KUKA KRL program: MyProgram_281().src

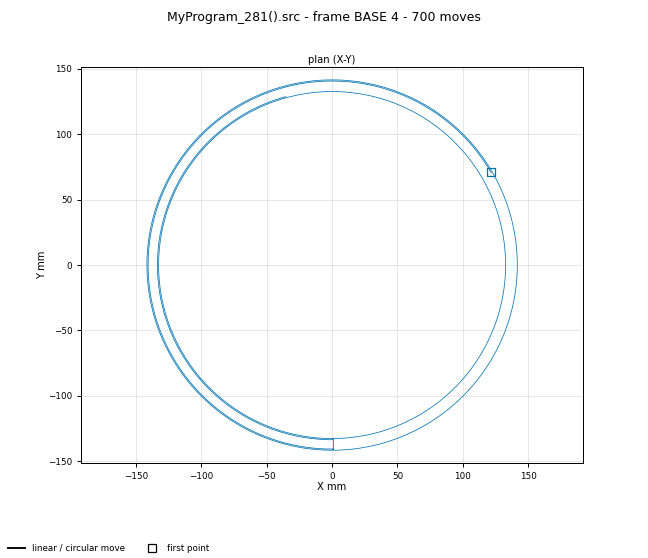
[picture p0: tool path of MyProgram_281().src in frame BASE 4, 700 of 700 moves have a stored position in this frame; points joined in program order, loops and branches not executed]
&ACCESS RVP
&REL 1
&PARAM TEMPLATE = C:\KRC\Roboter\Template\vorgabe
&PARAM EDITMASK = *
DEF MyProgram_281()
; ---- Setting reference (Base) ----
$BASE = BASE_DATA[4]

; --------------------------
; ---- Setting tool (TCP) ----
$TOOL = TOOL_DATA[3]
; --------------------------

$VEL.CP = VEL_APROX_PRINT
Startdeposition()
$VEL.CP = VEL_PRINT
LIN {X 121.5397,Y 70.8644,Z 173,A 32.0171,B 8.0887,C 0.1794,E1 8.2284,E2 419.8054} C_DIS
LIN {X 119.2507,Y 74.6518,Z 173,A 33.7721,B 8.0887,C 0.176,E1 8.2258,E2 418.0556} C_DIS
LIN {X 116.9146,Y 78.2591,Z 173,A 35.5172,B 8.0888,C 0.1719,E1 8.2231,E2 416.3103} C_DIS
LIN {X 114.3453,Y 81.9674,Z 173,A 37.3012,B 8.0889,C 0.1687,E1 8.2202,E2 414.5323} C_DIS
LIN {X 111.9951,Y 85.1512,Z 173,A 39.575,B 8.0893,C 0.1513,E1 8.2163,E2 412.1717} C_DIS
LIN {X 108.1696,Y 89.9605,Z 173,A 41.4044,B 8.0891,C 0.1597,E1 8.2132,E2 410.4289} C_DIS
LIN {X 105.5546,Y 93.0147,Z 173,A 43.0233,B 8.0891,C 0.1566,E1 8.2102,E2 408.8119} C_DIS
LIN {X 102.1646,Y 96.7261,Z 173,A 44.9523,B 8.0891,C 0.1547,E1 8.2066,E2 406.8974} C_DIS
LIN {X 99.1597,Y 99.804,Z 173,A 46.5834,B 8.0892,C 0.1536,E1 8.2034,E2 405.2813} C_DIS
LIN {X 93.6633,Y 104.9796,Z 173,A 49.7603,B 8.0894,C 0.1456,E1 8.1969,E2 402.0906} C_DIS
LIN {X 90.2461,Y 107.9313,Z 173,A 51.5389,B 8.0894,C 0.1434,E1 8.1931,E2 400.3193} C_DIS
LIN {X 86.802,Y 110.7199,Z 173,A 53.3455,B 8.0894,C 0.1401,E1 8.1891,E2 398.5122} C_DIS
LIN {X 83.1158,Y 113.5134,Z 173,A 55.2323,B 8.0895,C 0.1368,E1 8.1849,E2 396.6246} C_DIS
LIN {X 79.1384,Y 116.3216,Z 173,A 57.1673,B 8.0895,C 0.1345,E1 8.1805,E2 394.6955} C_DIS
LIN {X 75.4314,Y 118.7592,Z 173,A 58.9862,B 8.0895,C 0.1315,E1 8.1762,E2 392.8748} C_DIS
LIN {X 71.5988,Y 121.1084,Z 173,A 60.8066,B 8.0896,C 0.129,E1 8.1718,E2 391.0557} C_DIS
LIN {X 67.7143,Y 123.3224,Z 173,A 62.4595,B 8.0896,C 0.1297,E1 8.1679,E2 389.4242} C_DIS
LIN {X 62.8759,Y 125.8572,Z 173,A 64.811,B 8.0897,C 0.1244,E1 8.162,E2 387.0565} C_DIS
LIN {X 59.2274,Y 127.613,Z 173,A 66.3529,B 8.0897,C 0.1244,E1 8.1581,E2 385.5283} C_DIS
LIN {X 55.8685,Y 129.1187,Z 173,A 67.9786,B 8.0897,C 0.1202,E1 8.1539,E2 383.8865} C_DIS
LIN {X 51.5879,Y 130.8895,Z 173,A 69.7454,B 8.0897,C 0.1205,E1 8.1494,E2 382.1352} C_DIS
LIN {X 48.0453,Y 132.2298,Z 173,A 71.184,B 8.0897,C 0.121,E1 8.1457,E2 380.71} C_DIS
LIN {X 44.5635,Y 133.4431,Z 173,A 72.7767,B 8.0898,C 0.1179,E1 8.1414,E2 379.106} C_DIS
LIN {X 41.2024,Y 134.5189,Z 173,A 74.1193,B 8.0898,C 0.1184,E1 8.1379,E2 377.7757} C_DIS
LIN {X 38.0254,Y 135.4513,Z 173,A 75.499,B 8.0898,C 0.1168,E1 8.1342,E2 376.3921} C_DIS
LIN {X 35.189,Y 136.217,Z 173,A 77.1535,B 8.09,C 0.1073,E1 8.1296,E2 374.6794} C_DIS
LIN {X 31.0744,Y 137.2131,Z 173,A 78.431,B 8.0899,C 0.1146,E1 8.1262,E2 373.4594} C_DIS
LIN {X 27.0733,Y 138.0597,Z 173,A 80.1396,B 8.0899,C 0.1129,E1 8.1215,E2 371.7459} C_DIS
LIN {X 23.5323,Y 138.7061,Z 173,A 81.6734,B 8.0899,C 0.1109,E1 8.1173,E2 370.2038} C_DIS
LIN {X 18.8429,Y 139.4213,Z 173,A 83.3498,B 8.0899,C 0.1148,E1 8.1127,E2 368.5606} C_DIS
LIN {X 15.7013,Y 139.8103,Z 173,A 84.6671,B 8.0899,C 0.1139,E1 8.1091,E2 367.2401} C_DIS
LIN {X 12.7325,Y 140.1122,Z 173,A 86.1282,B 8.0899,C 0.1091,E1 8.1049,E2 365.7483} C_DIS
LIN {X 7.9682,Y 140.4636,Z 173,A 87.8716,B 8.0899,C 0.1124,E1 8.1001,E2 364.0314} C_DIS
LIN {X 4.257,Y 140.6239,Z 173,A 89.3394,B 8.0899,C 0.1131,E1 8.0961,E2 362.5699} C_DIS
LIN {X 1.4394,Y 140.6821,Z 173,A 90.4859,B 8.0899,C 0.1131,E1 8.0929,E2 361.4241} C_DIS
LIN {X -2.2697,Y 140.6696,Z 173,A 91.9938,B 8.0899,C 0.1131,E1 8.0887,E2 359.9172} C_DIS
LIN {X -5.6115,Y 140.5759,Z 173,A 93.5151,B 8.0899,C 0.1104,E1 8.0844,E2 358.3762} C_DIS
LIN {X -9.3168,Y 140.3806,Z 173,A 94.9136,B 8.0899,C 0.1127,E1 8.0805,E2 356.9929} C_DIS
LIN {X -12.9669,Y 140.0897,Z 173,A 96.3139,B 8.0899,C 0.1147,E1 8.0766,E2 355.6048} C_DIS
LIN {X -16.4487,Y 139.723,Z 173,A 97.8535,B 8.0899,C 0.1131,E1 8.0723,E2 354.0516} C_DIS
LIN {X -20.196,Y 139.2309,Z 173,A 99.5893,B 8.0899,C 0.1103,E1 8.0675,E2 352.2917} C_DIS
LIN {X -26.297,Y 138.2081,Z 173,A 102.423,B 8.0899,C 0.1062,E1 8.0596,E2 349.4193} C_DIS
LIN {X -30.692,Y 137.3005,Z 173,A 103.8767,B 8.0899,C 0.1138,E1 8.0557,E2 348.0146} C_DIS
LIN {X -35.3761,Y 136.1695,Z 173,A 105.8869,B 8.0899,C 0.1144,E1 8.0503,E2 345.9996} C_DIS
LIN {X -39.8029,Y 134.9399,Z 173,A 107.6544,B 8.0899,C 0.1176,E1 8.0456,E2 344.2465} C_DIS
LIN {X -44.0839,Y 133.6028,Z 173,A 109.4479,B 8.0898,C 0.1198,E1 8.0408,E2 342.4584} C_DIS
LIN {X -47.929,Y 132.2717,Z 173,A 111.3832,B 8.0898,C 0.1168,E1 8.0356,E2 340.4889} C_DIS
LIN {X -51.7917,Y 130.8101,Z 173,A 112.8658,B 8.0898,C 0.1219,E1 8.0318,E2 339.0331} C_DIS
LIN {X -55.5091,Y 129.2741,Z 173,A 114.4912,B 8.0898,C 0.124,E1 8.0277,E2 337.4105} C_DIS
LIN {X -61.4365,Y 126.5671,Z 173,A 117.2281,B 8.0897,C 0.1259,E1 8.0207,E2 334.6653} C_DIS
LIN {X -65.0696,Y 124.7357,Z 173,A 118.8403,B 8.0897,C 0.1288,E1 8.0167,E2 333.0599} C_DIS
LIN {X -68.2489,Y 123.0268,Z 173,A 120.467,B 8.0897,C 0.1283,E1 8.0127,E2 331.4146} C_DIS
LIN {X -72.3988,Y 120.632,Z 173,A 122.4005,B 8.0897,C 0.1315,E1 8.0081,E2 329.4851} C_DIS
LIN {X -76.3232,Y 118.1879,Z 173,A 124.3082,B 8.0896,C 0.134,E1 8.0036,E2 327.5758} C_DIS
LIN {X -80.2438,Y 115.5613,Z 173,A 126.0393,B 8.0895,C 0.1402,E1 7.9996,E2 325.8706} C_DIS
LIN {X -84.9117,Y 112.1763,Z 173,A 129.2567,B 8.0896,C 0.1303,E1 7.9922,E2 322.5441} C_DIS
LIN {X -89.5623,Y 108.4994,Z 173,A 130.8771,B 8.0893,C 0.1475,E1 7.9889,E2 321.0277} C_DIS
LIN {X -92.9813,Y 105.5841,Z 173,A 132.9319,B 8.0893,C 0.1475,E1 7.9845,E2 318.9459} C_DIS
LIN {X -95.7766,Y 103.055,Z 173,A 134.6016,B 8.0893,C 0.1483,E1 7.981,E2 317.2605} C_DIS
LIN {X -99.701,Y 99.2633,Z 173,A 136.5293,B 8.0891,C 0.1575,E1 7.9773,E2 315.3724} C_DIS
LIN {X -104.3128,Y 94.4052,Z 173,A 139.3278,B 8.0891,C 0.1622,E1 7.9719,E2 312.5678} C_DIS
LIN {X -109.1757,Y 88.7372,Z 173,A 142.5436,B 8.089,C 0.1663,E1 7.9661,E2 309.3328} C_DIS
LIN {X -111.9882,Y 85.1602,Z 173,A 144.3871,B 8.0889,C 0.1707,E1 7.9629,E2 307.4923} C_DIS
LIN {X -114.5373,Y 81.699,Z 173,A 146.118,B 8.0888,C 0.1751,E1 7.9601,E2 305.7656} C_DIS
LIN {X -116.8361,Y 78.3766,Z 173,A 147.8453,B 8.0888,C 0.1778,E1 7.9574,E2 304.0296} C_DIS
LIN {X -120.2813,Y 72.9789,Z 173,A 150.5347,B 8.0886,C 0.183,E1 7.9534,E2 301.3323} C_DIS
LIN {X -122.903,Y 68.4723,Z 173,A 152.688,B 8.0885,C 0.1879,E1 7.9504,E2 299.1773} C_DIS
LIN {X -125.091,Y 64.386,Z 173,A 154.5092,B 8.0884,C 0.1937,E1 7.948,E2 297.3665} C_DIS
LIN {X -126.5803,Y 61.4089,Z 173,A 156.0139,B 8.0884,C 0.195,E1 7.9462,E2 295.8442} C_DIS
LIN {X -128.0317,Y 58.3219,Z 173,A 157.4645,B 8.0883,C 0.1978,E1 7.9445,E2 294.3871} C_DIS
LIN {X -129.6212,Y 54.695,Z 173,A 158.9373,B 8.0881,C 0.2042,E1 7.9429,E2 292.9338} C_DIS
LIN {X -130.9965,Y 51.3126,Z 173,A 160.2682,B 8.0879,C 0.2105,E1 7.9415,E2 291.6243} C_DIS
LIN {X -132.2272,Y 48.0524,Z 173,A 161.9677,B 8.0879,C 0.2102,E1 7.9398,E2 289.8903} C_DIS
LIN {X -133.4973,Y 44.4008,Z 173,A 163.4771,B 8.0879,C 0.2155,E1 7.9385,E2 288.3909} C_DIS
LIN {X -134.5688,Y 41.0391,Z 173,A 164.8901,B 8.0877,C 0.2198,E1 7.9373,E2 286.9823} C_DIS
LIN {X -135.4878,Y 37.8948,Z 173,A 166.2428,B 8.0877,C 0.2233,E1 7.9363,E2 285.6285} C_DIS
LIN {X -136.2722,Y 34.9715,Z 173,A 167.6133,B 8.0876,C 0.2246,E1 7.9353,E2 284.2416} C_DIS
LIN {X -137.0675,Y 31.7118,Z 173,A 169.0149,B 8.0875,C 0.228,E1 7.9344,E2 282.8367} C_DIS
LIN {X -138.4552,Y 24.9642,Z 173,A 171.7558,B 8.0872,C 0.2369,E1 7.9329,E2 280.1069} C_DIS
LIN {X -139.392,Y 19.0614,Z 173,A 174.3063,B 8.0871,C 0.2422,E1 7.9318,E2 277.5439} C_DIS
LIN {X -139.9884,Y 14.0225,Z 173,A 176.6134,B 8.087,C 0.2445,E1 7.9311,E2 275.2077} C_DIS
LIN {X -140.3173,Y 10.2038,Z 173,A 178.5693,B 8.087,C 0.243,E1 7.9307,E2 273.2019} C_DIS
LIN {X -140.5888,Y 5.2818,Z 173,A -179.9247,B 8.0866,C 0.2564,E1 7.9305,E2 271.7629} C_DIS
LIN {X -140.6787,Y -1.7183,Z 173,A -176.9036,B 8.0864,C 0.2621,E1 7.9305,E2 268.7225} C_DIS
LIN {X -140.5167,Y -6.9375,Z 173,A -174.8865,B 8.0862,C 0.2698,E1 7.9307,E2 266.7214} C_DIS
LIN {X -140.2633,Y -10.9436,Z 173,A -173.1133,B 8.0862,C 0.2725,E1 7.9311,E2 264.9317} C_DIS
LIN {X -139.341,Y -19.4256,Z 173,A -169.8202,B 8.0857,C 0.2852,E1 7.9321,E2 261.6652} C_DIS
LIN {X -138.8167,Y -22.8693,Z 173,A -168.246,B 8.0857,C 0.2868,E1 7.9328,E2 260.072} C_DIS
LIN {X -138.2199,Y -26.2355,Z 173,A -166.7828,B 8.0855,C 0.2897,E1 7.9336,E2 258.6007} C_DIS
LIN {X -137.4925,Y -29.8133,Z 173,A -165.3249,B 8.0853,C 0.2943,E1 7.9344,E2 257.1477} C_DIS
LIN {X -136.7395,Y -33.0954,Z 173,A -163.9364,B 8.0853,C 0.2979,E1 7.9353,E2 255.7579} C_DIS
LIN {X -135.9183,Y -36.3208,Z 173,A -162.5627,B 8.0851,C 0.3014,E1 7.9363,E2 254.3829} C_DIS
LIN {X -134.9268,Y -39.8475,Z 173,A -161.0054,B 8.085,C 0.3045,E1 7.9375,E2 252.8183} C_DIS
LIN {X -133.6154,Y -44.0459,Z 173,A -159.2293,B 8.0848,C 0.3096,E1 7.939,E2 251.0454} C_DIS
LIN {X -132.2087,Y -48.1038,Z 173,A -157.2964,B 8.0848,C 0.3115,E1 7.9408,E2 249.0898} C_DIS
LIN {X -130.5376,Y -52.468,Z 173,A -155.6934,B 8.0843,C 0.3212,E1 7.9424,E2 247.5271} C_DIS
LIN {X -129.2717,Y -55.5146,Z 173,A -154.1083,B 8.0843,C 0.321,E1 7.9441,E2 245.9115} C_DIS
LIN {X -127.8562,Y -58.7014,Z 173,A -152.6637,B 8.0843,C 0.3243,E1 7.9458,E2 244.4646} C_DIS
LIN {X -126.333,Y -61.9114,Z 173,A -151.2786,B 8.084,C 0.3289,E1 7.9475,E2 243.0884} C_DIS
LIN {X -124.5763,Y -65.3731,Z 173,A -148.4644,B 8.0846,C 0.3135,E1 7.9514,E2 240.1127} C_DIS
LIN {X -120.64,Y -72.3853,Z 173,A -146.1641,B 8.0837,C 0.337,E1 7.9544,E2 237.9432} C_DIS
LIN {X -117.8769,Y -76.8022,Z 173,A -144.0223,B 8.0835,C 0.3417,E1 7.9576,E2 235.7998} C_DIS
LIN {X -115.2733,Y -80.6578,Z 173,A -142.085,B 8.0833,C 0.3454,E1 7.9607,E2 233.8579} C_DIS
LIN {X -112.6344,Y -84.3036,Z 173,A -140.2391,B 8.0832,C 0.3494,E1 7.9638,E2 232.0111} C_DIS
LIN {X -109.7952,Y -87.9698,Z 173,A -138.3153,B 8.083,C 0.353,E1 7.9671,E2 230.0834} C_DIS
LIN {X -106.8869,Y -91.4814,Z 173,A -136.1315,B 8.083,C 0.3517,E1 7.9711,E2 227.8573} C_DIS
LIN {X -104.2877,Y -94.4328,Z 173,A -134.8234,B 8.0827,C 0.3598,E1 7.9735,E2 226.5884} C_DIS
LIN {X -101.5037,Y -97.4195,Z 173,A -133.1573,B 8.0826,C 0.3631,E1 7.9767,E2 224.9224} C_DIS
LIN {X -98.6922,Y -100.2665,Z 173,A -131.3687,B 8.0826,C 0.3637,E1 7.9803,E2 223.1134} C_DIS
LIN {X -94.8602,Y -103.9,Z 173,A -129.2725,B 8.0823,C 0.3686,E1 7.9846,E2 221.025} C_DIS
LIN {X -91.3696,Y -106.9821,Z 173,A -127.3587,B 8.0822,C 0.3718,E1 7.9886,E2 219.1092} C_DIS
LIN {X -87.741,Y -109.9773,Z 173,A -125.4408,B 8.082,C 0.3751,E1 7.9928,E2 217.1915} C_DIS
LIN {X -83.5306,Y -113.2086,Z 173,A -123.1789,B 8.082,C 0.377,E1 7.9978,E2 214.9167} C_DIS
LIN {X -79.4321,Y -116.1209,Z 173,A -121.217,B 8.0817,C 0.3816,E1 8.0023,E2 212.9664} C_DIS
LIN {X -75.8907,Y -118.4655,Z 173,A -119.466,B 8.0817,C 0.3838,E1 8.0064,E2 211.2128} C_DIS
LIN {X -71.8963,Y -120.9315,Z 173,A -117.5578,B 8.0815,C 0.3865,E1 8.011,E2 209.3051} C_DIS
LIN {X -69.3467,Y -122.412,Z 173,A -115.7889,B 8.0819,C 0.3784,E1 8.0155,E2 207.4609} C_DIS
LIN {X -64.8654,Y -124.8429,Z 173,A -114.2083,B 8.0813,C 0.3895,E1 8.0192,E2 205.9462} C_DIS
LIN {X -61.0098,Y -126.771,Z 173,A -112.5189,B 8.0812,C 0.3927,E1 8.0234,E2 204.2655} C_DIS
LIN {X -56.6312,Y -128.7889,Z 173,A -110.574,B 8.0811,C 0.3952,E1 8.0284,E2 202.323} C_DIS
LIN {X -53.3702,Y -130.1739,Z 173,A -108.9867,B 8.0811,C 0.3941,E1 8.0325,E2 200.7165} C_DIS
LIN {X -49.8269,Y -131.5693,Z 173,A -107.6282,B 8.0809,C 0.3989,E1 8.036,E2 199.3831} C_DIS
LIN {X -46.9077,Y -132.6399,Z 173,A -106.18,B 8.0809,C 0.3968,E1 8.0398,E2 197.9108} C_DIS
LIN {X -43.0184,Y -133.9493,Z 173,A -104.614,B 8.0809,C 0.4,E1 8.044,E2 196.3583} C_DIS
LIN {X -38.913,Y -135.2004,Z 173,A -102.5335,B 8.0811,C 0.3952,E1 8.0497,E2 194.2334} C_DIS
LIN {X -35.4651,Y -136.1465,Z 173,A -101.3993,B 8.0807,C 0.4019,E1 8.0526,E2 193.1416} C_DIS
LIN {X -31.503,Y -137.1152,Z 173,A -99.6866,B 8.0807,C 0.4019,E1 8.0573,E2 191.4217} C_DIS
LIN {X -28.5134,Y -137.7687,Z 173,A -98.4424,B 8.0807,C 0.4026,E1 8.0607,E2 190.1774} C_DIS
LIN {X -25.6225,Y -138.3364,Z 173,A -97.109,B 8.0808,C 0.4006,E1 8.0644,E2 188.826} C_DIS
LIN {X -21.893,Y -138.9743,Z 173,A -95.8468,B 8.0805,C 0.4062,E1 8.0678,E2 187.6003} C_DIS
LIN {X -18.5725,Y -139.4567,Z 173,A -94.2702,B 8.0807,C 0.4028,E1 8.0722,E2 185.9953} C_DIS
LIN {X -14.0852,Y -139.9824,Z 173,A -92.475,B 8.0807,C 0.404,E1 8.0772,E2 184.2054} C_DIS
LIN {X -10.485,Y -140.2967,Z 173,A -90.9975,B 8.0807,C 0.404,E1 8.0813,E2 182.7265} C_DIS
LIN {X -6.2607,Y -140.5505,Z 173,A -89.1335,B 8.0807,C 0.4014,E1 8.0865,E2 180.8431} C_DIS
LIN {X -1.5063,Y -140.6817,Z 173,A -87.3668,B 8.0807,C 0.4045,E1 8.0914,E2 179.0982} C_DIS
LIN {X 0.9966,Y -140.684,Z 173,A -86.7203,B 8.0803,C 0.4113,E1 8.0931,E2 178.5006} C_DIS
Enddeposition()
LIN {X 0.9966,Y -140.684,Z 173,A -86.7203,B 8.0803,C 0.4113,E1 8.0931,E2 178.5006} C_DIS
Startdeposition()
$VEL.CP = VEL_PRINT
LIN {X 0.0008,Y -141.5985,Z 173,A -87.3284,B 8.0796,C 0.42,E1 8.091,E2 179.1698} C_DIS
LIN {X -2.9523,Y -141.5669,Z 173,A -88.5344,B 8.0796,C 0.4203,E1 8.0877,E2 180.3779} C_DIS
LIN {X -6.4248,Y -141.4522,Z 173,A -90.091,B 8.0795,C 0.4231,E1 8.0833,E2 181.9551} C_DIS
LIN {X -10.4048,Y -141.2135,Z 173,A -91.574,B 8.0796,C 0.4205,E1 8.0792,E2 183.4214} C_DIS
LIN {X -13.8781,Y -140.915,Z 173,A -92.979,B 8.0796,C 0.4202,E1 8.0753,E2 184.8262} C_DIS
LIN {X -17.1895,Y -140.5496,Z 173,A -94.3385,B 8.0796,C 0.4202,E1 8.0715,E2 186.1877} C_DIS
LIN {X -20.7709,Y -140.0665,Z 173,A -95.7933,B 8.0796,C 0.4196,E1 8.0675,E2 187.642} C_DIS
LIN {X -24.2041,Y -139.5142,Z 173,A -97.2155,B 8.0796,C 0.4194,E1 8.0635,E2 189.0667} C_DIS
LIN {X -27.6244,Y -138.8767,Z 173,A -98.6204,B 8.0797,C 0.4187,E1 8.0597,E2 190.4716} C_DIS
LIN {X -31.0173,Y -138.1581,Z 173,A -99.9098,B 8.0798,C 0.416,E1 8.0562,E2 191.7464} C_DIS
LIN {X -33.8951,Y -137.4813,Z 173,A -101.2277,B 8.0798,C 0.4175,E1 8.0526,E2 193.0806} C_DIS
LIN {X -37.2579,Y -136.6086,Z 173,A -102.6325,B 8.0798,C 0.4166,E1 8.0488,E2 194.4856} C_DIS
LIN {X -40.3664,Y -135.7216,Z 173,A -104.1154,B 8.0798,C 0.4188,E1 8.0448,E2 195.9918} C_DIS
LIN {X -44.9118,Y -134.2847,Z 173,A -105.97,B 8.0798,C 0.416,E1 8.0399,E2 197.837} C_DIS
LIN {X -48.8467,Y -132.9065,Z 173,A -107.5933,B 8.08,C 0.4134,E1 8.0356,E2 199.4522} C_DIS
LIN {X -52.0928,Y -131.668,Z 173,A -109.0108,B 8.08,C 0.4123,E1 8.0319,E2 200.8713} C_DIS
LIN {X -56.2644,Y -129.9373,Z 173,A -110.896,B 8.08,C 0.4114,E1 8.027,E2 202.7642} C_DIS
LIN {X -59.7557,Y -128.3697,Z 173,A -112.4081,B 8.0802,C 0.4091,E1 8.0232,E2 204.2716} C_DIS
LIN {X -63.4258,Y -126.599,Z 173,A -114.0734,B 8.0802,C 0.4075,E1 8.019,E2 205.9391} C_DIS
LIN {X -66.7353,Y -124.8858,Z 173,A -115.6997,B 8.0802,C 0.4076,E1 8.015,E2 207.5811} C_DIS
LIN {X -70.5472,Y -122.7731,Z 173,A -117.4889,B 8.0804,C 0.4057,E1 8.0106,E2 209.3736} C_DIS
LIN {X -74.5003,Y -120.415,Z 173,A -119.3629,B 8.0804,C 0.4033,E1 8.0061,E2 211.2489} C_DIS
LIN {X -78.1616,Y -118.0713,Z 173,A -121.1386,B 8.0806,C 0.401,E1 8.002,E2 213.0266} C_DIS
LIN {X -82.0256,Y -115.4206,Z 173,A -123.0413,B 8.0807,C 0.3981,E1 7.9976,E2 214.9299} C_DIS
LIN {X -85.7396,Y -112.6889,Z 173,A -124.8747,B 8.0809,C 0.3945,E1 7.9935,E2 216.7588} C_DIS
LIN {X -89.1541,Y -110.0073,Z 173,A -126.7136,B 8.0809,C 0.3929,E1 7.9895,E2 218.6081} C_DIS
LIN {X -92.6824,Y -107.0516,Z 173,A -128.5779,B 8.0812,C 0.3896,E1 7.9855,E2 220.4723} C_DIS
LIN {X -96.1818,Y -103.9191,Z 173,A -130.4624,B 8.0813,C 0.3858,E1 7.9816,E2 222.3542} C_DIS
LIN {X -99.3281,Y -100.9155,Z 173,A -132.2779,B 8.0815,C 0.3833,E1 7.978,E2 224.1765} C_DIS
LIN {X -102.5166,Y -97.6746,Z 173,A -134.0126,B 8.0817,C 0.3779,E1 7.9746,E2 225.8968} C_DIS
LIN {X -104.91,Y -95.0991,Z 173,A -135.5902,B 8.0817,C 0.3775,E1 7.9716,E2 227.4942} C_DIS
LIN {X -107.9521,Y -91.6313,Z 173,A -137.4853,B 8.0819,C 0.374,E1 7.9681,E2 229.3923} C_DIS
LIN {X -110.9324,Y -88,Z 173,A -139.3449,B 8.0821,C 0.3692,E1 7.9649,E2 231.2458} C_DIS
LIN {X -113.578,Y -84.5575,Z 173,A -141.1682,B 8.0822,C 0.3663,E1 7.9618,E2 233.077} C_DIS
LIN {X -116.2656,Y -80.8224,Z 173,A -143.0817,B 8.0824,C 0.3628,E1 7.9587,E2 234.9964} C_DIS
LIN {X -118.6886,Y -77.2204,Z 173,A -144.8629,B 8.0826,C 0.3591,E1 7.956,E2 236.7799} C_DIS
LIN {X -121.136,Y -73.3214,Z 173,A -146.749,B 8.0827,C 0.355,E1 7.9532,E2 238.668} C_DIS
LIN {X -123.4918,Y -69.2801,Z 173,A -148.6629,B 8.0829,C 0.3506,E1 7.9505,E2 240.5836} C_DIS
LIN {X -125.567,Y -65.4406,Z 173,A -150.397,B 8.0831,C 0.3457,E1 7.9483,E2 242.3126} C_DIS
LIN {X -126.9801,Y -62.6533,Z 173,A -151.7113,B 8.0832,C 0.3433,E1 7.9466,E2 243.6326} C_DIS
LIN {X -128.6243,Y -59.205,Z 173,A -153.2596,B 8.0834,C 0.3393,E1 7.9448,E2 245.1802} C_DIS
LIN {X -130.1442,Y -55.7861,Z 173,A -154.7693,B 8.0836,C 0.3353,E1 7.9431,E2 246.6885} C_DIS
LIN {X -131.4752,Y -52.5722,Z 173,A -156.1988,B 8.0837,C 0.3319,E1 7.9416,E2 248.1199} C_DIS
LIN {X -132.7228,Y -49.3375,Z 173,A -157.6704,B 8.0838,C 0.3292,E1 7.9401,E2 249.5994} C_DIS
LIN {X -134.2854,Y -44.9097,Z 173,A -159.5572,B 8.084,C 0.3239,E1 7.9384,E2 251.4832} C_DIS
LIN {X -135.3463,Y -41.6032,Z 173,A -161.0737,B 8.0841,C 0.3217,E1 7.9371,E2 253.0131} C_DIS
LIN {X -136.4655,Y -37.7722,Z 173,A -162.6285,B 8.0843,C 0.3164,E1 7.9359,E2 254.559} C_DIS
LIN {X -137.3538,Y -34.4031,Z 173,A -164.062,B 8.0845,C 0.3128,E1 7.9349,E2 255.9945} C_DIS
LIN {X -138.1566,Y -31.0238,Z 173,A -165.4411,B 8.0846,C 0.3085,E1 7.9341,E2 257.369} C_DIS
LIN {X -138.7726,Y -28.1359,Z 173,A -166.711,B 8.0847,C 0.3063,E1 7.9334,E2 258.6477} C_DIS
LIN {X -139.4213,Y -24.7232,Z 173,A -168.1406,B 8.0849,C 0.3027,E1 7.9326,E2 260.0793} C_DIS
LIN {X -139.987,Y -21.2903,Z 173,A -169.5528,B 8.0849,C 0.2987,E1 7.932,E2 261.491} C_DIS
LIN {X -140.4695,Y -17.8361,Z 173,A -171.0016,B 8.0851,C 0.2953,E1 7.9315,E2 262.9435} C_DIS
LIN {X -140.865,Y -14.3923,Z 173,A -172.4437,B 8.0852,C 0.2919,E1 7.931,E2 264.3895} C_DIS
LIN {X -141.1748,Y -10.9356,Z 173,A -173.9987,B 8.0853,C 0.2901,E1 7.9307,E2 265.9627} C_DIS
LIN {X -141.425,Y -6.9652,Z 173,A -175.5055,B 8.0855,C 0.2839,E1 7.9304,E2 267.4548} C_DIS
LIN {X -141.5537,Y -3.5022,Z 173,A -176.9238,B 8.0857,C 0.2801,E1 7.9304,E2 268.8739} C_DIS
LIN {X -141.5999,Y -0.016,Z 173,A -178.3743,B 8.0857,C 0.2766,E1 7.9303,E2 270.3284} C_DIS
LIN {X -141.5207,Y 4.6893,Z 173,A 179.6709,B 8.0859,C 0.2719,E1 7.9304,E2 272.2879} C_DIS
LIN {X -141.3313,Y 8.6596,Z 173,A 178.0397,B 8.0861,C 0.2676,E1 7.9307,E2 273.9205} C_DIS
LIN {X -141.0751,Y 12.1397,Z 173,A 176.6126,B 8.0862,C 0.2637,E1 7.931,E2 275.3483} C_DIS
LIN {X -140.7367,Y 15.5848,Z 173,A 175.187,B 8.0863,C 0.2601,E1 7.9314,E2 276.7757} C_DIS
LIN {X -140.3111,Y 19.0453,Z 173,A 173.7549,B 8.0864,C 0.2564,E1 7.9319,E2 278.2092} C_DIS
LIN {X -139.8046,Y 22.468,Z 173,A 172.3118,B 8.0865,C 0.253,E1 7.9325,E2 279.6566} C_DIS
LIN {X -139.2133,Y 25.8774,Z 173,A 170.8827,B 8.0867,C 0.2494,E1 7.9332,E2 281.0881} C_DIS
LIN {X -138.5378,Y 29.2766,Z 173,A 169.5536,B 8.0868,C 0.2444,E1 7.9339,E2 282.4064} C_DIS
LIN {X -137.8858,Y 32.2095,Z 173,A 168.2359,B 8.0868,C 0.2425,E1 7.9348,E2 283.736} C_DIS
LIN {X -137.0534,Y 35.5868,Z 173,A 166.7963,B 8.087,C 0.239,E1 7.9358,E2 285.1784} C_DIS
LIN {X -136.1394,Y 38.9383,Z 173,A 165.2183,B 8.087,C 0.2376,E1 7.937,E2 286.777} C_DIS
LIN {X -135.0545,Y 42.5444,Z 173,A 163.6509,B 8.0871,C 0.2341,E1 7.9383,E2 288.3484} C_DIS
LIN {X -133.4964,Y 47.2108,Z 173,A 161.7841,B 8.0873,C 0.2268,E1 7.9399,E2 290.1975} C_DIS
LIN {X -132.2979,Y 50.4719,Z 173,A 160.351,B 8.0874,C 0.2233,E1 7.9413,E2 291.6327} C_DIS
LIN {X -131.0192,Y 53.7033,Z 173,A 158.6858,B 8.0874,C 0.2234,E1 7.9431,E2 293.3294} C_DIS
LIN {X -129.0903,Y 58.1828,Z 173,A 156.8718,B 8.0876,C 0.2158,E1 7.9451,E2 295.1212} C_DIS
LIN {X -127.2479,Y 62.1104,Z 173,A 155.23,B 8.0878,C 0.2095,E1 7.9471,E2 296.7467} C_DIS
LIN {X -125.9654,Y 64.6709,Z 173,A 153.8757,B 8.0878,C 0.2095,E1 7.9488,E2 298.1247} C_DIS
LIN {X -123.7569,Y 68.8059,Z 173,A 151.9893,B 8.0879,C 0.2044,E1 7.9513,E2 300.008} C_DIS
LIN {X -121.5879,Y 72.5696,Z 173,A 150.1547,B 8.0879,C 0.2012,E1 7.9539,E2 301.8506} C_DIS
LIN {X -119.1717,Y 76.4728,Z 173,A 148.31,B 8.0881,C 0.1964,E1 7.9567,E2 303.6918} C_DIS
LIN {X -116.7581,Y 80.1093,Z 173,A 146.46,B 8.0881,C 0.1934,E1 7.9596,E2 305.5507} C_DIS
LIN {X -114.0944,Y 83.8595,Z 173,A 144.5675,B 8.0883,C 0.1895,E1 7.9627,E2 307.4453} C_DIS
LIN {X -111.4706,Y 87.3171,Z 173,A 142.783,B 8.0883,C 0.1859,E1 7.9657,E2 309.2317} C_DIS
LIN {X -108.5516,Y 90.9203,Z 173,A 140.8956,B 8.0884,C 0.1819,E1 7.9691,E2 311.1186} C_DIS
LIN {X -105.5581,Y 94.3792,Z 173,A 139.0023,B 8.0885,C 0.1785,E1 7.9726,E2 313.0156} C_DIS
LIN {X -102.6012,Y 97.5862,Z 173,A 137.1886,B 8.0885,C 0.1755,E1 7.976,E2 314.8337} C_DIS
LIN {X -99.515,Y 100.7316,Z 173,A 135.4599,B 8.0887,C 0.171,E1 7.9794,E2 316.5539} C_DIS
LIN {X -96.5769,Y 103.5512,Z 173,A 133.7939,B 8.0887,C 0.1679,E1 7.9828,E2 318.2206} C_DIS
LIN {X -93.3587,Y 106.4622,Z 173,A 131.9544,B 8.0887,C 0.1659,E1 7.9867,E2 320.069} C_DIS
LIN {X -89.8361,Y 109.4509,Z 173,A 130.0589,B 8.0888,C 0.1628,E1 7.9907,E2 321.9661} C_DIS
LIN {X -86.4521,Y 112.1433,Z 173,A 128.2813,B 8.0889,C 0.1601,E1 7.9946,E2 323.7456} C_DIS
LIN {X -82.7628,Y 114.8931,Z 173,A 126.3907,B 8.0889,C 0.1573,E1 7.9989,E2 325.6382} C_DIS
LIN {X -78.8844,Y 117.5895,Z 173,A 124.5314,B 8.089,C 0.1534,E1 8.0032,E2 327.4893} C_DIS
LIN {X -75.2389,Y 119.9551,Z 173,A 122.7046,B 8.089,C 0.1517,E1 8.0075,E2 329.3232} C_DIS
LIN {X -71.3046,Y 122.3347,Z 173,A 120.8109,B 8.0891,C 0.1495,E1 8.012,E2 331.2195} C_DIS
LIN {X -67.2852,Y 124.5903,Z 173,A 118.946,B 8.0891,C 0.1469,E1 8.0166,E2 333.0828} C_DIS
LIN {X -63.6672,Y 126.4763,Z 173,A 117.431,B 8.0892,C 0.1424,E1 8.0203,E2 334.5793} C_DIS
LIN {X -60.7819,Y 127.8867,Z 173,A 116.0719,B 8.0892,C 0.1418,E1 8.0238,E2 335.9449} C_DIS
LIN {X -57.6143,Y 129.3446,Z 173,A 114.6219,B 8.0892,C 0.1407,E1 8.0274,E2 337.3988} C_DIS
LIN {X -54.1942,Y 130.8149,Z 173,A 113.1381,B 8.0892,C 0.1386,E1 8.0313,E2 338.8786} C_DIS
LIN {X -50.978,Y 132.1013,Z 173,A 111.6788,B 8.0893,C 0.1381,E1 8.0351,E2 340.3441} C_DIS
LIN {X -47.2193,Y 133.4934,Z 173,A 109.9184,B 8.0893,C 0.1388,E1 8.0397,E2 342.1209} C_DIS
LIN {X -43.26,Y 134.8259,Z 173,A 108.3938,B 8.0893,C 0.1345,E1 8.0437,E2 343.6233} C_DIS
LIN {X -39.4413,Y 135.9924,Z 173,A 106.771,B 8.0893,C 0.1332,E1 8.0481,E2 345.2458} C_DIS
LIN {X -36.0943,Y 136.9189,Z 173,A 105.2913,B 8.0893,C 0.1334,E1 8.0521,E2 346.7341} C_DIS
LIN {X -31.8757,Y 137.962,Z 173,A 103.5209,B 8.0894,C 0.1324,E1 8.0569,E2 348.5048} C_DIS
LIN {X -28.1671,Y 138.7663,Z 173,A 102.052,B 8.0894,C 0.1304,E1 8.0609,E2 349.9643} C_DIS
LIN {X -24.7634,Y 139.4141,Z 173,A 100.6464,B 8.0894,C 0.1297,E1 8.0647,E2 351.3696} C_DIS
LIN {X -21.3335,Y 139.9803,Z 173,A 99.2799,B 8.0894,C 0.1283,E1 8.0685,E2 352.7301} C_DIS
LIN {X -17.851,Y 140.4676,Z 173,A 97.8181,B 8.0894,C 0.1285,E1 8.0725,E2 354.1961} C_DIS
LIN {X -14.8389,Y 140.8169,Z 173,A 96.5366,B 8.0894,C 0.129,E1 8.0761,E2 355.4838} C_DIS
LIN {X -10.9413,Y 141.1744,Z 173,A 94.8643,B 8.0894,C 0.1302,E1 8.0808,E2 357.1666} C_DIS
LIN {X -6.9546,Y 141.4255,Z 173,A 93.3776,B 8.0894,C 0.1276,E1 8.0849,E2 358.636} C_DIS
LIN {X -3.4759,Y 141.5545,Z 173,A 91.9802,B 8.0894,C 0.1273,E1 8.0888,E2 360.0313} C_DIS
LIN {X -0.0037,Y 141.5985,Z 173,A 90.5893,B 8.0894,C 0.127,E1 8.0927,E2 361.4198} C_DIS
LIN {X 2.9503,Y 141.5669,Z 173,A 89.3828,B 8.0894,C 0.1272,E1 8.096,E2 362.6272} C_DIS
LIN {X 6.4229,Y 141.4523,Z 173,A 88.0062,B 8.0894,C 0.1268,E1 8.0999,E2 363.9995} C_DIS
LIN {X 10.4159,Y 141.2127,Z 173,A 86.3436,B 8.0894,C 0.1279,E1 8.1045,E2 365.667} C_DIS
LIN {X 13.8739,Y 140.9154,Z 173,A 84.9459,B 8.0894,C 0.1282,E1 8.1084,E2 367.0634} C_DIS
LIN {X 17.3249,Y 140.5335,Z 173,A 83.5468,B 8.0894,C 0.1285,E1 8.1123,E2 368.4612} C_DIS
LIN {X 20.7727,Y 140.0662,Z 173,A 82.141,B 8.0894,C 0.129,E1 8.1162,E2 369.8663} C_DIS
LIN {X 24.2085,Y 139.5134,Z 173,A 80.7176,B 8.0894,C 0.13,E1 8.1201,E2 371.2913} C_DIS
LIN {X 27.6173,Y 138.8781,Z 173,A 79.3225,B 8.0894,C 0.1306,E1 8.1239,E2 372.685} C_DIS
LIN {X 31.0091,Y 138.16,Z 173,A 78.0496,B 8.0894,C 0.129,E1 8.1273,E2 373.9409} C_DIS
LIN {X 33.8918,Y 137.4821,Z 173,A 76.7425,B 8.0894,C 0.1318,E1 8.1309,E2 375.2617} C_DIS
LIN {X 37.2334,Y 136.6152,Z 173,A 75.3502,B 8.0894,C 0.1328,E1 8.1347,E2 376.653} C_DIS
LIN {X 41.1056,Y 135.4986,Z 173,A 73.7236,B 8.0894,C 0.134,E1 8.139,E2 378.2788} C_DIS
LIN {X 44.9102,Y 134.2852,Z 173,A 72.0442,B 8.0894,C 0.1366,E1 8.1435,E2 379.966} C_DIS
LIN {X 48.8461,Y 132.9067,Z 173,A 70.4393,B 8.0894,C 0.1366,E1 8.1477,E2 381.5602} C_DIS
LIN {X 52.0935,Y 131.6677,Z 173,A 69.0389,B 8.0894,C 0.138,E1 8.1514,E2 382.9598} C_DIS
LIN {X 55.2644,Y 130.368,Z 173,A 67.6052,B 8.0893,C 0.1404,E1 8.1551,E2 384.3993} C_DIS
LIN {X 58.1475,Y 129.1061,Z 173,A 66.396,B 8.0893,C 0.1407,E1 8.1581,E2 385.6002} C_DIS
LIN {X 61.3132,Y 127.6329,Z 173,A 64.9404,B 8.0893,C 0.1432,E1 8.1618,E2 387.0612} C_DIS
LIN {X 65.1957,Y 125.6957,Z 173,A 63.1609,B 8.0892,C 0.146,E1 8.1663,E2 388.8438} C_DIS
LIN {X 69.2618,Y 123.5021,Z 173,A 61.3074,B 8.0892,C 0.1482,E1 8.1708,E2 390.6953} C_DIS
LIN {X 73.3198,Y 121.1369,Z 173,A 59.4409,B 8.0891,C 0.1503,E1 8.1753,E2 392.5576} C_DIS
LIN {X 76.997,Y 118.8336,Z 173,A 57.6959,B 8.0891,C 0.1528,E1 8.1794,E2 394.3013} C_DIS
LIN {X 80.815,Y 116.2707,Z 173,A 55.8446,B 8.089,C 0.1556,E1 8.1836,E2 396.1517} C_DIS
LIN {X 84.5584,Y 113.5774,Z 173,A 53.9974,B 8.089,C 0.1584,E1 8.1878,E2 397.9968} C_DIS
LIN {X 88.0013,Y 110.9314,Z 173,A 52.2498,B 8.0889,C 0.1613,E1 8.1916,E2 399.7435} C_DIS
LIN {X 91.6265,Y 107.9562,Z 173,A 50.438,B 8.0889,C 0.1631,E1 8.1955,E2 401.5448} C_DIS
LIN {X 94.8379,Y 105.147,Z 173,A 48.7244,B 8.0888,C 0.1661,E1 8.1991,E2 403.2571} C_DIS
LIN {X 98.0085,Y 102.1975,Z 173,A 47.0248,B 8.0888,C 0.1685,E1 8.2025,E2 404.9505} C_DIS
LIN {X 100.7366,Y 99.5101,Z 173,A 45.4619,B 8.0887,C 0.1719,E1 8.2056,E2 406.5156} C_DIS
LIN {X 103.5606,Y 96.5668,Z 173,A 43.7986,B 8.0886,C 0.1756,E1 8.2088,E2 408.1811} C_DIS
LIN {X 106.6406,Y 93.1544,Z 173,A 41.9441,B 8.0885,C 0.1795,E1 8.2123,E2 410.0355} C_DIS
LIN {X 109.5062,Y 89.7685,Z 173,A 40.1682,B 8.0885,C 0.183,E1 8.2154,E2 411.8097} C_DIS
LIN {X 112.4634,Y 86.0345,Z 173,A 38.3566,B 8.0884,C 0.185,E1 8.2185,E2 413.6072} C_DIS
LIN {X 114.9114,Y 82.7375,Z 173,A 36.6167,B 8.0883,C 0.1904,E1 8.2214,E2 415.3579} C_DIS
LIN {X 117.5913,Y 78.8818,Z 173,A 34.8133,B 8.0882,C 0.1929,E1 8.2242,E2 417.1498} C_DIS
LIN {X 119.9533,Y 75.2417,Z 173,A 33.0329,B 8.0881,C 0.1977,E1 8.2269,E2 418.9342} C_DIS
LIN {X 122.3336,Y 71.3065,Z 173,A 31.1849,B 8.088,C 0.202,E1 8.2295,E2 420.7816} C_DIS
LIN {X 124.5907,Y 67.2844,Z 173,A 29.3643,B 8.0879,C 0.2058,E1 8.232,E2 422.5974} C_DIS
LIN {X 126.4775,Y 63.6649,Z 173,A 27.8401,B 8.0879,C 0.2073,E1 8.2339,E2 424.1061} C_DIS
LIN {X 128.0049,Y 60.5346,Z 173,A 26.3573,B 8.0877,C 0.2125,E1 8.2357,E2 425.5991} C_DIS
LIN {X 129.9343,Y 56.2714,Z 173,A 24.513,B 8.0877,C 0.2164,E1 8.2378,E2 427.4382} C_DIS
LIN {X 131.4657,Y 52.5955,Z 173,A 23.003,B 8.0875,C 0.2186,E1 8.2394,E2 428.9362} C_DIS
LIN {X 132.7224,Y 49.3384,Z 173,A 21.5724,B 8.0875,C 0.2227,E1 8.2408,E2 430.3701} C_DIS
LIN {X 134.285,Y 44.911,Z 173,A 19.7492,B 8.0873,C 0.2263,E1 8.2425,E2 432.1846} C_DIS
LIN {X 135.3462,Y 41.6036,Z 173,A 18.284,B 8.0872,C 0.2314,E1 8.2437,E2 433.6586} C_DIS
LIN {X 136.4681,Y 37.7631,Z 173,A 16.7782,B 8.0872,C 0.2335,E1 8.2448,E2 435.151} C_DIS
LIN {X 137.3585,Y 34.3844,Z 173,A 15.3905,B 8.087,C 0.2369,E1 8.2458,E2 436.5363} C_DIS
LIN {X 138.1594,Y 31.0115,Z 173,A 14.0601,B 8.087,C 0.2393,E1 8.2466,E2 437.8584} C_DIS
LIN {X 138.7737,Y 28.1309,Z 173,A 12.8391,B 8.0868,C 0.2432,E1 8.2473,E2 439.084} C_DIS
LIN {X 139.3908,Y 24.8932,Z 173,A 11.5045,B 8.0868,C 0.247,E1 8.248,E2 440.4198} C_DIS
LIN {X 139.9855,Y 21.3,Z 173,A 10.0861,B 8.0866,C 0.25,E1 8.2486,E2 441.8323} C_DIS
LIN {X 140.4663,Y 17.8607,Z 173,A 8.71,B 8.0866,C 0.2534,E1 8.2491,E2 443.2057} C_DIS
LIN {X 140.8645,Y 14.3964,Z 173,A 7.3124,B 8.0864,C 0.2572,E1 8.2496,E2 444.6029} C_DIS
LIN {X 141.1747,Y 10.9366,Z 173,A 5.8101,B 8.0862,C 0.2633,E1 8.2499,E2 446.1189} C_DIS
LIN {X 141.4255,Y 6.9545,Z 173,A 4.3526,B 8.0862,C 0.2646,E1 8.2501,E2 447.5573} C_DIS
LIN {X 141.5542,Y 3.4847,Z 173,A 2.8703,B 8.086,C 0.2703,E1 8.2503,E2 449.051} C_DIS
LIN {X 141.5957,Y -0.7174,Z 173,A 1.2301,B 8.0859,C 0.2739,E1 8.2503,E2 450.6848} C_DIS
LIN {X 141.5207,Y -4.6903,Z 173,A -0.2955,B 8.0858,C 0.2768,E1 8.2502,E2 452.2012} C_DIS
LIN {X 141.3677,Y -8.0688,Z 173,A -1.7661,B 8.0856,C 0.283,E1 8.2499,E2 453.6863} C_DIS
LIN {X 141.0747,Y -12.1452,Z 173,A -3.2472,B 8.0856,C 0.284,E1 8.2496,E2 455.1464} C_DIS
LIN {X 140.7341,Y -15.6089,Z 173,A -4.6256,B 8.0854,C 0.2874,E1 8.2492,E2 456.5222} C_DIS
LIN {X 140.3099,Y -19.0538,Z 173,A -6.003,B 8.0853,C 0.2909,E1 8.2487,E2 457.8975} C_DIS
LIN {X 139.8013,Y -22.4888,Z 173,A -7.4056,B 8.0851,C 0.2949,E1 8.2481,E2 459.301} C_DIS
LIN {X 139.2074,Y -25.9084,Z 173,A -8.7833,B 8.0851,C 0.2983,E1 8.2475,E2 460.6766} C_DIS
LIN {X 138.6684,Y -28.6479,Z 173,A -9.8961,B 8.0849,C 0.3012,E1 8.2468,E2 461.7882} C_DIS
LIN {X 137.8864,Y -32.2065,Z 173,A -11.3281,B 8.0848,C 0.3045,E1 8.246,E2 463.2162} C_DIS
LIN {X 137.056,Y -35.5765,Z 173,A -12.7094,B 8.0847,C 0.3079,E1 8.245,E2 464.5958} C_DIS
LIN {X 136.1424,Y -38.9276,Z 173,A -14.2231,B 8.0844,C 0.3142,E1 8.2439,E2 466.1251} C_DIS
LIN {X 135.0248,Y -42.6375,Z 173,A -15.7647,B 8.0843,C 0.318,E1 8.2426,E2 467.6648} C_DIS
LIN {X 133.4962,Y -47.2113,Z 173,A -17.5546,B 8.0842,C 0.3199,E1 8.241,E2 469.4354} C_DIS
LIN {X 132.2963,Y -50.476,Z 173,A -18.9396,B 8.0841,C 0.3233,E1 8.2396,E2 470.819} C_DIS
LIN {X 131.0182,Y -53.7059,Z 173,A -20.5457,B 8.0837,C 0.3314,E1 8.2379,E2 472.4528} C_DIS
LIN {X 129.0978,Y -58.1662,Z 173,A -22.2551,B 8.0837,C 0.3312,E1 8.236,E2 474.1305} C_DIS
LIN {X 127.6337,Y -61.3116,Z 173,A -23.6902,B 8.0836,C 0.3356,E1 8.2343,E2 475.5712} C_DIS
LIN {X 125.7117,Y -65.1652,Z 173,A -25.4552,B 8.0834,C 0.3406,E1 8.2321,E2 477.3409} C_DIS
LIN {X 123.4998,Y -69.2658,Z 173,A -27.298,B 8.0832,C 0.3446,E1 8.2296,E2 479.1801} C_DIS
LIN {X 121.1392,Y -73.316,Z 173,A -29.1526,B 8.083,C 0.3485,E1 8.227,E2 481.031} C_DIS
LIN {X 118.8297,Y -77.003,Z 173,A -30.8871,B 8.0829,C 0.3523,E1 8.2244,E2 482.7639} C_DIS
LIN {X 116.2746,Y -80.8094,Z 173,A -32.7227,B 8.0827,C 0.3564,E1 8.2215,E2 484.5988} C_DIS
LIN {X 113.5927,Y -84.5379,Z 173,A -34.5545,B 8.0825,C 0.3603,E1 8.2185,E2 486.4289} C_DIS
LIN {X 110.9488,Y -87.9794,Z 173,A -36.3033,B 8.0823,C 0.3643,E1 8.2155,E2 488.1785} C_DIS
LIN {X 108.0432,Y -91.5242,Z 173,A -38.0946,B 8.0822,C 0.3672,E1 8.2123,E2 489.9633} C_DIS
LIN {X 105.0971,Y -94.8929,Z 173,A -39.8593,B 8.0821,C 0.3703,E1 8.209,E2 491.7237} C_DIS
LIN {X 102.1393,Y -98.0694,Z 173,A -41.5822,B 8.0819,C 0.3734,E1 8.2057,E2 493.4439} C_DIS
LIN {X 99.3241,Y -100.9194,Z 173,A -43.2451,B 8.0817,C 0.3777,E1 8.2024,E2 495.1139} C_DIS
LIN {X 96.1843,Y -103.9168,Z 173,A -44.9937,B 8.0816,C 0.3811,E1 8.1988,E2 496.8631} C_DIS
LIN {X 92.6912,Y -107.044,Z 173,A -46.8512,B 8.0814,C 0.3841,E1 8.195,E2 498.7171} C_DIS
LIN {X 89.1563,Y -110.0055,Z 173,A -48.7037,B 8.0813,C 0.3874,E1 8.191,E2 500.5697} C_DIS
LIN {X 85.7439,Y -112.6856,Z 173,A -50.4422,B 8.0811,C 0.3903,E1 8.1871,E2 502.3074} C_DIS
LIN {X 82.2509,Y -115.2595,Z 173,A -52.1665,B 8.081,C 0.3928,E1 8.1832,E2 504.0292} C_DIS
LIN {X 78.8832,Y -117.5903,Z 173,A -53.7541,B 8.081,C 0.3942,E1 8.1796,E2 505.6091} C_DIS
LIN {X 75.2475,Y -119.9496,Z 173,A -55.5403,B 8.0808,C 0.3978,E1 8.1754,E2 507.4012} C_DIS
LIN {X 71.3168,Y -122.3277,Z 173,A -57.3987,B 8.0806,C 0.4007,E1 8.1709,E2 509.261} C_DIS
LIN {X 67.2883,Y -124.5886,Z 173,A -59.234,B 8.0806,C 0.4028,E1 8.1664,E2 511.0934} C_DIS
LIN {X 63.6652,Y -126.4774,Z 173,A -60.7754,B 8.0806,C 0.4028,E1 8.1626,E2 512.6214} C_DIS
LIN {X 60.5414,Y -128.0017,Z 173,A -62.2591,B 8.0803,C 0.4063,E1 8.1589,E2 514.1164} C_DIS
LIN {X 56.2818,Y -129.9298,Z 173,A -64.1233,B 8.0803,C 0.4082,E1 8.1541,E2 515.9784} C_DIS
LIN {X 52.5796,Y -131.4722,Z 173,A -65.6525,B 8.0803,C 0.4082,E1 8.1502,E2 517.4965} C_DIS
LIN {X 49.3421,Y -132.7211,Z 173,A -67.0906,B 8.0801,C 0.4105,E1 8.1464,E2 518.9402} C_DIS
LIN {X 44.9193,Y -134.2822,Z 173,A -68.9306,B 8.0801,C 0.4114,E1 8.1416,E2 520.7739} C_DIS
LIN {X 41.6018,Y -135.3468,Z 173,A -70.4163,B 8.0799,C 0.4143,E1 8.1376,E2 522.2707} C_DIS
LIN {X 37.7687,Y -136.4665,Z 173,A -71.9384,B 8.0799,C 0.4139,E1 8.1335,E2 523.7815} C_DIS
LIN {X 34.3942,Y -137.3561,Z 173,A -73.3396,B 8.0799,C 0.4149,E1 8.1297,E2 525.1822} C_DIS
LIN {X 31.0215,Y -138.1571,Z 173,A -74.6857,B 8.0799,C 0.4149,E1 8.1261,E2 526.5217} C_DIS
LIN {X 28.1381,Y -138.7722,Z 173,A -75.9252,B 8.0799,C 0.4166,E1 8.1227,E2 527.7681} C_DIS
LIN {X 24.7294,Y -139.4201,Z 173,A -77.3215,B 8.0798,C 0.4174,E1 8.1188,E2 529.1643} C_DIS
LIN {X 21.3039,Y -139.9849,Z 173,A -78.7181,B 8.0798,C 0.418,E1 8.115,E2 530.5607} C_DIS
LIN {X 17.8626,Y -140.466,Z 173,A -80.1158,B 8.0798,C 0.4186,E1 8.1111,E2 531.9581} C_DIS
LIN {X 14.3981,Y -140.8644,Z 173,A -81.5336,B 8.0797,C 0.4193,E1 8.1072,E2 533.3777} C_DIS
LIN {X 10.9385,Y -141.1746,Z 173,A -83.0598,B 8.0795,C 0.4221,E1 8.1029,E2 534.9206} C_DIS
LIN {X 6.9583,Y -141.4254,Z 173,A -84.5416,B 8.0796,C 0.42,E1 8.0988,E2 536.3858} C_DIS
LIN {X 3.5575,Y -141.5522,Z 173,A -85.9138,B 8.0796,C 0.4202,E1 8.095,E2 537.758} C_DIS
LIN {X 1.0025,Y -141.5919,Z 173,A -86.6713,B 8.0799,C 0.4152,E1 8.093,E2 538.4792} C_DIS
Enddeposition()
LIN {X 0.9609,Y -132.6531,Z 174,A -86.8217,B 7.8952,C 0.3729,E1 7.9067,E2 538.3641} C_DIS
Startdeposition()
$VEL.CP = VEL_PRINT
LIN {X 3.5384,Y -132.6117,Z 174,A -85.4392,B 7.8955,C 0.3681,E1 7.9107,E2 536.9479} C_DIS
LIN {X 6.5007,Y -132.4995,Z 174,A -84.1106,B 7.8955,C 0.367,E1 7.9144,E2 535.6127} C_DIS
LIN {X 9.7566,Y -132.2995,Z 174,A -82.7613,B 7.8955,C 0.3676,E1 7.9182,E2 534.27} C_DIS
LIN {X 13.5559,Y -131.9658,Z 174,A -81.1804,B 7.8955,C 0.3681,E1 7.9225,E2 532.6965} C_DIS
LIN {X 16.9055,Y -131.5775,Z 174,A -79.8457,B 7.8954,C 0.3695,E1 7.9262,E2 531.376} C_DIS
LIN {X 19.4578,Y -131.2258,Z 174,A -78.4735,B 7.8956,C 0.3644,E1 7.9301,E2 529.971} C_DIS
LIN {X 22.9482,Y -130.6594,Z 174,A -77.1207,B 7.8956,C 0.3666,E1 7.9338,E2 528.6389} C_DIS
LIN {X 26.1646,Y -130.0531,Z 174,A -75.6205,B 7.8956,C 0.3641,E1 7.9379,E2 527.1271} C_DIS
LIN {X 29.0672,Y -129.4358,Z 174,A -74.273,B 7.8957,C 0.362,E1 7.9416,E2 525.7706} C_DIS
LIN {X 32.5097,Y -128.6134,Z 174,A -72.8269,B 7.8957,C 0.3622,E1 7.9455,E2 524.3337} C_DIS
LIN {X 35.6508,Y -127.7783,Z 174,A -71.431,B 7.8957,C 0.3611,E1 7.9493,E2 522.9378} C_DIS
LIN {X 39.3639,Y -126.6849,Z 174,A -69.609,B 7.896,C 0.3568,E1 7.9542,E2 521.096} C_DIS
LIN {X 43.4371,Y -125.3454,Z 174,A -67.9306,B 7.896,C 0.358,E1 7.9586,E2 519.4378} C_DIS
LIN {X 46.4958,Y -124.2432,Z 174,A -66.6072,B 7.896,C 0.358,E1 7.962,E2 518.1232} C_DIS
LIN {X 49.2601,Y -123.1739,Z 174,A -65.199,B 7.896,C 0.3541,E1 7.9657,E2 516.6982} C_DIS
LIN {X 52.5282,Y -121.8156,Z 174,A -63.7504,B 7.8961,C 0.3537,E1 7.9694,E2 515.2584} C_DIS
LIN {X 55.2378,Y -120.6119,Z 174,A -62.4842,B 7.8961,C 0.3523,E1 7.9726,E2 513.993} C_DIS
LIN {X 58.4338,Y -119.0957,Z 174,A -60.9597,B 7.8963,C 0.3503,E1 7.9765,E2 512.4676} C_DIS
LIN {X 61.3534,Y -117.6185,Z 174,A -59.6166,B 7.8963,C 0.3496,E1 7.9798,E2 511.1321} C_DIS
LIN {X 64.1418,Y -116.1232,Z 174,A -58.2767,B 7.8963,C 0.3481,E1 7.9831,E2 509.7944} C_DIS
LIN {X 66.7445,Y -114.6474,Z 174,A -56.9304,B 7.8965,C 0.3451,E1 7.9864,E2 508.4403} C_DIS
LIN {X 69.4956,Y -113.0006,Z 174,A -55.4972,B 7.8966,C 0.342,E1 7.9898,E2 506.9998} C_DIS
LIN {X 73.0679,Y -110.7242,Z 174,A -53.8777,B 7.8966,C 0.3429,E1 7.9935,E2 505.4048} C_DIS
LIN {X 75.0508,Y -109.3898,Z 174,A -52.6532,B 7.8968,C 0.3375,E1 7.9964,E2 504.1556} C_DIS
LIN {X 77.7176,Y -107.5116,Z 174,A -51.3426,B 7.8968,C 0.3368,E1 7.9994,E2 502.8559} C_DIS
LIN {X 80.8479,Y -105.1783,Z 174,A -49.6486,B 7.897,C 0.3336,E1 8.0032,E2 501.1594} C_DIS
LIN {X 84.0476,Y -102.639,Z 174,A -47.8822,B 7.8971,C 0.3302,E1 8.007,E2 499.3911} C_DIS
LIN {X 87.2606,Y -99.9216,Z 174,A -46.0051,B 7.8973,C 0.3255,E1 8.011,E2 497.5049} C_DIS
LIN {X 90.3246,Y -97.1608,Z 174,A -44.2828,B 7.8974,C 0.323,E1 8.0145,E2 495.7882} C_DIS
LIN {X 92.558,Y -95.0364,Z 174,A -42.9023,B 7.8976,C 0.3193,E1 8.0173,E2 494.4004} C_DIS
LIN {X 95.6132,Y -91.9622,Z 174,A -41.0747,B 7.8976,C 0.3162,E1 8.0209,E2 492.5766} C_DIS
LIN {X 98.3947,Y -88.9791,Z 174,A -39.3603,B 7.8978,C 0.3132,E1 8.0241,E2 490.8663} C_DIS
LIN {X 101.3796,Y -85.5632,Z 174,A -37.4681,B 7.8979,C 0.3101,E1 8.0275,E2 488.9804} C_DIS
LIN {X 104.0784,Y -82.2594,Z 174,A -35.699,B 7.898,C 0.3073,E1 8.0306,E2 487.2186} C_DIS
LIN {X 106.5557,Y -79.0234,Z 174,A -33.9536,B 7.8982,C 0.3034,E1 8.0335,E2 485.4733} C_DIS
LIN {X 108.765,Y -75.9538,Z 174,A -32.4826,B 7.8982,C 0.3026,E1 8.0359,E2 484.0208} C_DIS
LIN {X 110.4637,Y -73.4615,Z 174,A -31.1547,B 7.8984,C 0.299,E1 8.038,E2 482.6884} C_DIS
LIN {X 112.2359,Y -70.7238,Z 174,A -29.7192,B 7.8985,C 0.2949,E1 8.0401,E2 481.2482} C_DIS
LIN {X 113.9345,Y -67.9536,Z 174,A -28.3321,B 7.8986,C 0.2917,E1 8.0421,E2 479.8617} C_DIS
LIN {X 115.5801,Y -65.1154,Z 174,A -27.0164,B 7.8986,C 0.2901,E1 8.0439,E2 478.5571} C_DIS
LIN {X 116.9988,Y -62.531,Z 174,A -25.6698,B 7.8989,C 0.2854,E1 8.0458,E2 477.2002} C_DIS
LIN {X 118.4918,Y -59.6513,Z 174,A -24.2958,B 7.8989,C 0.2822,E1 8.0475,E2 475.8282} C_DIS
LIN {X 120.0296,Y -56.4952,Z 174,A -22.823,B 7.8991,C 0.2791,E1 8.0493,E2 474.3592} C_DIS
LIN {X 121.26,Y -53.7995,Z 174,A -21.5588,B 7.8991,C 0.276,E1 8.0507,E2 473.0956} C_DIS
LIN {X 122.6727,Y -50.4984,Z 174,A -20.0384,B 7.8993,C 0.2724,E1 8.0524,E2 471.5775} C_DIS
LIN {X 123.7686,Y -47.7461,Z 174,A -18.7834,B 7.8994,C 0.2694,E1 8.0536,E2 470.3241} C_DIS
LIN {X 124.9019,Y -44.6973,Z 174,A -17.3754,B 7.8995,C 0.2655,E1 8.055,E2 468.9144} C_DIS
LIN {X 126.1735,Y -40.9746,Z 174,A -15.7632,B 7.8996,C 0.2625,E1 8.0564,E2 467.3113} C_DIS
LIN {X 127.3232,Y -37.2432,Z 174,A -14.037,B 7.8998,C 0.257,E1 8.0578,E2 465.5785} C_DIS
LIN {X 128.2656,Y -33.8575,Z 174,A -12.5923,B 7.8999,C 0.2542,E1 8.0588,E2 464.1413} C_DIS
LIN {X 129.1004,Y -30.5237,Z 174,A -11.1518,B 7.9,C 0.2509,E1 8.0598,E2 462.7047} C_DIS
LIN {X 129.7876,Y -27.4551,Z 174,A -9.7649,B 7.9002,C 0.2465,E1 8.0606,E2 461.3131} C_DIS
LIN {X 130.4186,Y -24.2835,Z 174,A -8.4035,B 7.9002,C 0.2432,E1 8.0613,E2 459.9547} C_DIS
LIN {X 131.0216,Y -20.7823,Z 174,A -6.9107,B 7.9004,C 0.2396,E1 8.062,E2 458.4655} C_DIS
LIN {X 131.491,Y -17.5658,Z 174,A -5.5342,B 7.9004,C 0.2361,E1 8.0625,E2 457.091} C_DIS
LIN {X 131.9263,Y -13.9235,Z 174,A -4.0523,B 7.9005,C 0.2336,E1 8.063,E2 455.6202} C_DIS
LIN {X 132.1934,Y -11.1018,Z 174,A -2.8379,B 7.9006,C 0.2303,E1 8.0633,E2 454.4058} C_DIS
LIN {X 132.4274,Y -7.8379,Z 174,A -1.4394,B 7.9008,C 0.2265,E1 8.0636,E2 453.0079} C_DIS
LIN {X 132.5694,Y -4.8791,Z 174,A -0.1515,B 7.9008,C 0.2226,E1 8.0637,E2 451.7178} C_DIS
LIN {X 132.6543,Y -1.2569,Z 174,A 1.2235,B 7.9008,C 0.2219,E1 8.0637,E2 450.3647} C_DIS
LIN {X 132.6455,Y 1.9089,Z 174,A 2.7477,B 7.9011,C 0.2148,E1 8.0637,E2 448.8201} C_DIS
LIN {X 132.5585,Y 5.1584,Z 174,A 4.1585,B 7.9011,C 0.2106,E1 8.0637,E2 447.4072} C_DIS
LIN {X 132.3912,Y 8.4261,Z 174,A 5.5202,B 7.9013,C 0.2076,E1 8.0634,E2 446.0507} C_DIS
LIN {X 132.048,Y 12.7143,Z 174,A 7.3658,B 7.9013,C 0.2025,E1 8.0629,E2 444.2049} C_DIS
LIN {X 131.6629,Y 16.2319,Z 174,A 8.8183,B 7.9015,C 0.1997,E1 8.0625,E2 442.7605} C_DIS
LIN {X 131.178,Y 19.772,Z 174,A 10.3489,B 7.9015,C 0.1955,E1 8.0619,E2 441.2302} C_DIS
LIN {X 130.656,Y 22.9672,Z 174,A 11.6301,B 7.9016,C 0.1938,E1 8.0613,E2 439.9621} C_DIS
LIN {X 130.0538,Y 26.1608,Z 174,A 13.1006,B 7.9017,C 0.1886,E1 8.0605,E2 438.4824} C_DIS
LIN {X 129.4365,Y 29.0639,Z 174,A 14.4332,B 7.9018,C 0.184,E1 8.0597,E2 437.1427} C_DIS
LIN {X 128.6113,Y 32.5181,Z 174,A 15.8635,B 7.9019,C 0.1817,E1 8.0587,E2 435.7238} C_DIS
LIN {X 127.7752,Y 35.662,Z 174,A 17.2435,B 7.9019,C 0.1783,E1 8.0577,E2 434.3459} C_DIS
LIN {X 126.8558,Y 38.8056,Z 174,A 18.6316,B 7.9021,C 0.1749,E1 8.0566,E2 432.9599} C_DIS
LIN {X 125.7327,Y 42.3049,Z 174,A 20.2283,B 7.9021,C 0.1704,E1 8.0552,E2 431.3611} C_DIS
LIN {X 124.2522,Y 46.472,Z 174,A 21.9966,B 7.9022,C 0.1681,E1 8.0536,E2 429.6087} C_DIS
LIN {X 123.0543,Y 49.5568,Z 174,A 23.467,B 7.9022,C 0.1634,E1 8.052,E2 428.1323} C_DIS
LIN {X 121.8127,Y 52.5348,Z 174,A 24.844,B 7.9024,C 0.1601,E1 8.0505,E2 426.7564} C_DIS
LIN {X 120.6096,Y 55.2429,Z 174,A 26.0996,B 7.9024,C 0.1572,E1 8.0491,E2 425.5031} C_DIS
LIN {X 119.091,Y 58.4432,Z 174,A 27.6044,B 7.9024,C 0.1537,E1 8.0473,E2 424.0003} C_DIS
LIN {X 117.6192,Y 61.3519,Z 174,A 28.9491,B 7.9025,C 0.1514,E1 8.0456,E2 422.6625} C_DIS
LIN {X 116.2139,Y 63.9781,Z 174,A 30.254,B 7.9026,C 0.1478,E1 8.0438,E2 421.3548} C_DIS
LIN {X 114.6101,Y 66.809,Z 174,A 31.6473,B 7.9026,C 0.1445,E1 8.0419,E2 419.9621} C_DIS
LIN {X 112.9381,Y 69.5975,Z 174,A 33.0731,B 7.9027,C 0.1407,E1 8.0398,E2 418.5331} C_DIS
LIN {X 111.1996,Y 72.3424,Z 174,A 34.4505,B 7.9027,C 0.1378,E1 8.0377,E2 417.1581} C_DIS
LIN {X 109.3918,Y 75.0479,Z 174,A 35.789,B 7.9028,C 0.1357,E1 8.0356,E2 415.827} C_DIS
LIN {X 107.5075,Y 77.7233,Z 174,A 37.204,B 7.9028,C 0.1324,E1 8.0333,E2 414.4112} C_DIS
LIN {X 105.092,Y 80.9604,Z 174,A 39.0354,B 7.903,C 0.1268,E1 8.0302,E2 412.5686} C_DIS
LIN {X 102.4951,Y 84.2237,Z 174,A 40.81,B 7.903,C 0.1233,E1 8.0271,E2 410.7964} C_DIS
LIN {X 99.8224,Y 87.3743,Z 174,A 42.5669,B 7.903,C 0.1199,E1 8.0239,E2 409.0422} C_DIS
LIN {X 96.8512,Y 90.6571,Z 174,A 44.3871,B 7.9031,C 0.1176,E1 8.0205,E2 407.2325} C_DIS
LIN {X 94.1235,Y 93.4854,Z 174,A 45.8925,B 7.9031,C 0.1178,E1 8.0176,E2 405.7495} C_DIS
LIN {X 91.9616,Y 95.6138,Z 174,A 47.4319,B 7.9032,C 0.1109,E1 8.0145,E2 404.1823} C_DIS
LIN {X 88.5865,Y 98.7481,Z 174,A 49.3247,B 7.9032,C 0.1088,E1 8.0106,E2 402.3005} C_DIS
LIN {X 85.5222,Y 101.414,Z 174,A 51.0543,B 7.9032,C 0.106,E1 8.0069,E2 400.5735} C_DIS
LIN {X 82.2606,Y 104.0774,Z 174,A 52.8199,B 7.9032,C 0.1037,E1 8.0031,E2 398.8139} C_DIS
LIN {X 79.0205,Y 106.5579,Z 174,A 54.5725,B 7.9033,C 0.1009,E1 7.9992,E2 397.0622} C_DIS
LIN {X 76.1756,Y 108.6101,Z 174,A 55.9917,B 7.9033,C 0.1001,E1 7.996,E2 395.6542} C_DIS
LIN {X 73.459,Y 110.4653,Z 174,A 57.3872,B 7.9033,C 0.0983,E1 7.9928,E2 394.2616} C_DIS
LIN {X 70.7284,Y 112.233,Z 174,A 58.8273,B 7.9034,C 0.0955,E1 7.9894,E2 392.8172} C_DIS
LIN {X 67.9589,Y 113.9313,Z 174,A 60.2158,B 7.9034,C 0.0937,E1 7.986,E2 391.4303} C_DIS
LIN {X 65.1447,Y 115.5636,Z 174,A 61.5424,B 7.9034,C 0.0931,E1 7.9828,E2 390.1131} C_DIS
LIN {X 62.547,Y 116.9902,Z 174,A 63.0439,B 7.9034,C 0.0874,E1 7.9791,E2 388.5851} C_DIS
LIN {X 59.6377,Y 118.4987,Z 174,A 64.3077,B 7.9034,C 0.0883,E1 7.976,E2 387.3394} C_DIS
LIN {X 56.456,Y 120.0483,Z 174,A 65.8028,B 7.9035,C 0.087,E1 7.9722,E2 385.8484} C_DIS
LIN {X 53.7569,Y 121.2791,Z 174,A 67.072,B 7.9035,C 0.0857,E1 7.969,E2 384.5806} C_DIS
LIN {X 50.5027,Y 122.6709,Z 174,A 68.5908,B 7.9035,C 0.0842,E1 7.9651,E2 383.0632} C_DIS
LIN {X 47.7434,Y 123.7696,Z 174,A 69.8619,B 7.9035,C 0.083,E1 7.9618,E2 381.7935} C_DIS
LIN {X 44.6961,Y 124.9024,Z 174,A 71.3002,B 7.9035,C 0.0811,E1 7.958,E2 380.3513} C_DIS
LIN {X 41.018,Y 126.1596,Z 174,A 73.0975,B 7.9035,C 0.0775,E1 7.9532,E2 378.5402} C_DIS
LIN {X 36.9725,Y 127.4025,Z 174,A 74.7409,B 7.9035,C 0.0792,E1 7.9489,E2 376.9191} C_DIS
LIN {X 33.8592,Y 128.2651,Z 174,A 76.1287,B 7.9035,C 0.0783,E1 7.9451,E2 375.5325} C_DIS
LIN {X 29.9671,Y 129.2302,Z 174,A 77.989,B 7.9036,C 0.0749,E1 7.94,E2 373.6574} C_DIS
LIN {X 25.8777,Y 130.1114,Z 174,A 79.6487,B 7.9036,C 0.0764,E1 7.9355,E2 372.0156} C_DIS
LIN {X 22.6777,Y 130.7078,Z 174,A 81.1376,B 7.9036,C 0.0743,E1 7.9314,E2 370.5173} C_DIS
LIN {X 19.185,Y 131.2648,Z 174,A 82.5893,B 7.9036,C 0.0749,E1 7.9274,E2 369.0751} C_DIS
LIN {X 15.5065,Y 131.7495,Z 174,A 84.097,B 7.9036,C 0.0759,E1 7.9233,E2 367.5791} C_DIS
LIN {X 12.3477,Y 132.0832,Z 174,A 85.4945,B 7.9036,C 0.0751,E1 7.9194,E2 366.1791} C_DIS
LIN {X 9.7585,Y 132.2994,Z 174,A 86.7167,B 7.9036,C 0.0732,E1 7.916,E2 364.9454} C_DIS
LIN {X 6.5128,Y 132.4989,Z 174,A 88.0662,B 7.9036,C 0.0739,E1 7.9122,E2 363.6031} C_DIS
LIN {X 3.2641,Y 132.6194,Z 174,A 89.5103,B 7.9036,C 0.0731,E1 7.9082,E2 362.1548} C_DIS
LIN {X 0.0164,Y 132.6608,Z 174,A 90.9832,B 7.9036,C 0.072,E1 7.9041,E2 360.6742} C_DIS
LIN {X -3.5439,Y 132.6116,Z 174,A 92.421,B 7.9036,C 0.0737,E1 7.9001,E2 359.249} C_DIS
LIN {X -6.5062,Y 132.4993,Z 174,A 93.751,B 7.9036,C 0.0731,E1 7.8963,E2 357.9137} C_DIS
LIN {X -9.752,Y 132.2999,Z 174,A 95.1031,B 7.9036,C 0.0742,E1 7.8926,E2 356.5685} C_DIS
LIN {X -13.0004,Y 132.0206,Z 174,A 96.509,B 7.9036,C 0.0746,E1 7.8887,E2 355.1637} C_DIS
LIN {X -16.241,Y 131.6618,Z 174,A 97.9164,B 7.9036,C 0.0751,E1 7.8848,E2 353.7571} C_DIS
LIN {X -19.4633,Y 131.225,Z 174,A 99.4199,B 7.9036,C 0.0741,E1 7.8806,E2 352.2428} C_DIS
LIN {X -22.956,Y 130.658,Z 174,A 100.7796,B 7.9036,C 0.0775,E1 7.8769,E2 350.9039} C_DIS
LIN {X -26.1535,Y 130.0553,Z 174,A 102.2831,B 7.9036,C 0.0768,E1 7.8728,E2 349.3896} C_DIS
LIN {X -29.6611,Y 129.3001,Z 174,A 103.7735,B 7.9036,C 0.0787,E1 7.8687,E2 347.9071} C_DIS
LIN {X -32.5133,Y 128.6125,Z 174,A 105.1104,B 7.9036,C 0.0785,E1 7.8651,E2 346.5628} C_DIS
LIN {X -35.6831,Y 127.7693,Z 174,A 106.5325,B 7.9036,C 0.0795,E1 7.8612,E2 345.141} C_DIS
LIN {X -38.7947,Y 126.8591,Z 174,A 107.9405,B 7.9036,C 0.0805,E1 7.8575,E2 343.733} C_DIS
LIN {X -41.7289,Y 125.9245,Z 174,A 109.314,B 7.9036,C 0.081,E1 7.8538,E2 342.3553} C_DIS
LIN {X -45.354,Y 124.6652,Z 174,A 110.8865,B 7.9036,C 0.084,E1 7.8497,E2 340.7941} C_DIS
LIN {X -47.7233,Y 123.7774,Z 174,A 112.0439,B 7.9036,C 0.0841,E1 7.8467,E2 339.6298} C_DIS
LIN {X -50.9957,Y 122.465,Z 174,A 113.5896,B 7.9036,C 0.0854,E1 7.8427,E2 338.0825} C_DIS
LIN {X -54.0223,Y 121.1604,Z 174,A 114.9292,B 7.9035,C 0.0884,E1 7.8393,E2 336.754} C_DIS
LIN {X -56.7157,Y 119.9242,Z 174,A 116.3816,B 7.9035,C 0.0873,E1 7.8355,E2 335.2822} C_DIS
LIN {X -59.9103,Y 118.3599,Z 174,A 117.8507,B 7.9035,C 0.0903,E1 7.8319,E2 333.8223} C_DIS
LIN {X -62.7916,Y 116.8588,Z 174,A 119.2717,B 7.9035,C 0.092,E1 7.8284,E2 332.4003} C_DIS
LIN {X -65.384,Y 115.429,Z 174,A 120.563,B 7.9035,C 0.0936,E1 7.8252,E2 331.1086} C_DIS
LIN {X -68.1899,Y 113.7936,Z 174,A 121.9817,B 7.9035,C 0.0955,E1 7.8218,E2 329.6891} C_DIS
LIN {X -71.1952,Y 111.9381,Z 174,A 123.4837,B 7.9034,C 0.0982,E1 7.8183,E2 328.1912} C_DIS
LIN {X -74.019,Y 110.0914,Z 174,A 125.1391,B 7.9034,C 0.0976,E1 7.8144,E2 326.5137} C_DIS
LIN {X -77.7168,Y 107.5122,Z 174,A 126.9556,B 7.9034,C 0.1028,E1 7.8103,E2 324.7143} C_DIS
LIN {X -80.8585,Y 105.1702,Z 174,A 128.6951,B 7.9033,C 0.1051,E1 7.8064,E2 322.9707} C_DIS
LIN {X -84.0401,Y 102.6451,Z 174,A 130.4963,B 7.9033,C 0.1076,E1 7.8025,E2 321.1655} C_DIS
LIN {X -87.2725,Y 99.9113,Z 174,A 132.4255,B 7.9033,C 0.1096,E1 7.7984,E2 319.226} C_DIS
LIN {X -90.3937,Y 97.0965,Z 174,A 134.26,B 7.9032,C 0.1129,E1 7.7946,E2 317.3909} C_DIS
LIN {X -93.3218,Y 94.286,Z 174,A 136.0434,B 7.9032,C 0.116,E1 7.791,E2 315.6056} C_DIS
LIN {X -96.0778,Y 91.476,Z 174,A 137.6635,B 7.9031,C 0.1207,E1 7.7879,E2 313.9965} C_DIS
LIN {X -98.8407,Y 88.4832,Z 174,A 139.5467,B 7.9031,C 0.1227,E1 7.7843,E2 312.1003} C_DIS
LIN {X -101.5023,Y 85.417,Z 174,A 141.2302,B 7.903,C 0.1276,E1 7.7813,E2 310.4268} C_DIS
LIN {X -104.0802,Y 82.2571,Z 174,A 143.0238,B 7.9029,C 0.1311,E1 7.7782,E2 308.631} C_DIS
LIN {X -106.5555,Y 79.0237,Z 174,A 144.8208,B 7.9029,C 0.1347,E1 7.7751,E2 306.8312} C_DIS
LIN {X -108.6544,Y 76.1128,Z 174,A 146.314,B 7.9028,C 0.1391,E1 7.7727,E2 305.3463} C_DIS
LIN {X -110.4708,Y 73.4508,Z 174,A 147.7174,B 7.9028,C 0.1423,E1 7.7705,E2 303.9428} C_DIS
LIN {X -112.2255,Y 70.7404,Z 174,A 149.1777,B 7.9027,C 0.1448,E1 7.7683,E2 302.4761} C_DIS
LIN {X -113.9124,Y 67.9906,Z 174,A 150.5897,B 7.9026,C 0.148,E1 7.7663,E2 301.0632} C_DIS
LIN {X -115.5249,Y 65.2136,Z 174,A 151.9496,B 7.9026,C 0.1519,E1 7.7644,E2 299.7079} C_DIS
LIN {X -116.9974,Y 62.5335,Z 174,A 153.3728,B 7.9025,C 0.1539,E1 7.7625,E2 298.2737} C_DIS
LIN {X -118.4937,Y 59.6475,Z 174,A 154.7982,B 7.9025,C 0.1572,E1 7.7607,E2 296.8472} C_DIS
LIN {X -120.0419,Y 56.4695,Z 174,A 156.4932,B 7.9024,C 0.1589,E1 7.7586,E2 295.1337} C_DIS
LIN {X -121.9239,Y 52.2777,Z 174,A 158.3786,B 7.9023,C 0.1655,E1 7.7565,E2 293.262} C_DIS
LIN {X -123.2825,Y 48.9907,Z 174,A 160.0167,B 7.9022,C 0.1683,E1 7.7548,E2 291.6133} C_DIS
LIN {X -124.9068,Y 44.6839,Z 174,A 161.9661,B 7.9021,C 0.1742,E1 7.7529,E2 289.6704} C_DIS
LIN {X -125.9642,Y 41.6097,Z 174,A 163.4264,B 7.9021,C 0.1773,E1 7.7516,E2 288.2047} C_DIS
LIN {X -127.3276,Y 37.2282,Z 174,A 165.4283,B 7.9019,C 0.1825,E1 7.75,E2 286.2024} C_DIS
LIN {X -128.2758,Y 33.8191,Z 174,A 166.9383,B 7.9018,C 0.187,E1 7.7489,E2 284.696} C_DIS
LIN {X -129.1322,Y 30.392,Z 174,A 168.4819,B 7.9017,C 0.1911,E1 7.7479,E2 283.1518} C_DIS
LIN {X -129.7983,Y 27.4053,Z 174,A 169.8752,B 7.9017,C 0.1939,E1 7.7471,E2 281.7512} C_DIS
LIN {X -130.4207,Y 24.2725,Z 174,A 171.2373,B 7.9015,C 0.198,E1 7.7464,E2 280.3925} C_DIS
LIN {X -131.0214,Y 20.7834,Z 174,A 172.8139,B 7.9015,C 0.2018,E1 7.7456,E2 278.8116} C_DIS
LIN {X -131.4912,Y 17.5644,Z 174,A 174.2432,B 7.9013,C 0.2055,E1 7.7451,E2 277.3806} C_DIS
LIN {X -131.8817,Y 14.3379,Z 174,A 175.6699,B 7.9013,C 0.2092,E1 7.7446,E2 275.9525} C_DIS
LIN {X -132.1949,Y 11.0847,Z 174,A 177.0487,B 7.9011,C 0.2137,E1 7.7443,E2 274.579} C_DIS
LIN {X -132.4273,Y 7.8397,Z 174,A 178.4919,B 7.9011,C 0.2172,E1 7.744,E2 273.1324} C_DIS
LIN {X -132.5694,Y 4.8795,Z 174,A 179.8302,B 7.9009,C 0.2201,E1 7.7439,E2 271.7883} C_DIS
LIN {X -132.6543,Y 1.2556,Z 174,A -178.7429,B 7.9008,C 0.2265,E1 7.7438,E2 270.3795} C_DIS
LIN {X -132.6454,Y -1.9105,Z 174,A -177.1563,B 7.9008,C 0.2275,E1 7.7438,E2 268.7677} C_DIS
LIN {X -132.5578,Y -5.1771,Z 174,A -175.7887,B 7.9006,C 0.2321,E1 7.7439,E2 267.4065} C_DIS
LIN {X -132.3787,Y -8.6284,Z 174,A -174.2673,B 7.9005,C 0.2361,E1 7.7442,E2 265.883} C_DIS
LIN {X -132.1699,Y -11.3807,Z 174,A -173,B 7.9005,C 0.2385,E1 7.7445,E2 264.6076} C_DIS
LIN {X -131.8428,Y -14.6993,Z 174,A -171.5398,B 7.9003,C 0.2423,E1 7.7449,E2 263.1462} C_DIS
LIN {X -131.4523,Y -17.8606,Z 174,A -170.1372,B 7.9002,C 0.2459,E1 7.7454,E2 261.7415} C_DIS
LIN {X -130.9285,Y -21.3601,Z 174,A -168.5589,B 7.9001,C 0.2495,E1 7.7461,E2 260.1584} C_DIS
LIN {X -130.3348,Y -24.722,Z 174,A -167.0952,B 7.8999,C 0.2538,E1 7.7468,E2 258.6971} C_DIS
LIN {X -129.6206,Y -28.2284,Z 174,A -165.429,B 7.8999,C 0.2565,E1 7.7478,E2 257.0175} C_DIS
LIN {X -128.6232,Y -32.471,Z 174,A -163.5773,B 7.8997,C 0.2622,E1 7.749,E2 255.1708} C_DIS
LIN {X -127.8025,Y -35.5643,Z 174,A -162.1719,B 7.8995,C 0.2657,E1 7.75,E2 253.7637} C_DIS
LIN {X -126.8611,Y -38.7881,Z 174,A -160.6891,B 7.8995,C 0.2692,E1 7.7512,E2 252.2779} C_DIS
LIN {X -125.9635,Y -41.612,Z 174,A -159.3201,B 7.8993,C 0.2715,E1 7.7524,E2 250.899} C_DIS
LIN {X -124.8089,Y -44.9553,Z 174,A -157.8315,B 7.8992,C 0.2761,E1 7.7538,E2 249.4162} C_DIS
LIN {X -123.6905,Y -47.9471,Z 174,A -156.3904,B 7.8991,C 0.279,E1 7.7552,E2 247.9686} C_DIS
LIN {X -122.4482,Y -51.036,Z 174,A -154.9656,B 7.8989,C 0.2829,E1 7.7567,E2 246.5463} C_DIS
LIN {X -121.1611,Y -54.0208,Z 174,A -153.6156,B 7.8988,C 0.2873,E1 7.7583,E2 245.2037} C_DIS
LIN {X -119.9172,Y -56.7303,Z 174,A -152.2336,B 7.8988,C 0.2893,E1 7.7599,E2 243.811} C_DIS
LIN {X -118.3646,Y -59.9011,Z 174,A -150.6818,B 7.8986,C 0.2928,E1 7.7618,E2 242.2568} C_DIS
LIN {X -116.8684,Y -62.7737,Z 174,A -149.3305,B 7.8984,C 0.297,E1 7.7636,E2 240.9122} C_DIS
LIN {X -115.4423,Y -65.3606,Z 174,A -147.9529,B 7.8984,C 0.2988,E1 7.7655,E2 239.5228} C_DIS
LIN {X -113.6566,Y -68.4179,Z 174,A -146.4525,B 7.8982,C 0.3029,E1 7.7676,E2 238.0268} C_DIS
LIN {X -111.925,Y -71.2156,Z 174,A -144.9991,B 7.8981,C 0.3058,E1 7.7698,E2 236.5702} C_DIS
LIN {X -110.1361,Y -73.9521,Z 174,A -143.5652,B 7.898,C 0.3088,E1 7.772,E2 235.1343} C_DIS
LIN {X -108.1579,Y -76.8167,Z 174,A -142.0766,B 7.8978,C 0.3125,E1 7.7744,E2 233.6481} C_DIS
LIN {X -106.5575,Y -79.0209,Z 174,A -140.6794,B 7.8978,C 0.312,E1 7.7767,E2 232.2244} C_DIS
LIN {X -104.0913,Y -82.2429,Z 174,A -138.8866,B 7.8978,C 0.3153,E1 7.7798,E2 230.4275} C_DIS
LIN {X -101.4141,Y -85.5221,Z 174,A -137.032,B 7.8976,C 0.3189,E1 7.7831,E2 228.5703} C_DIS
LIN {X -98.3931,Y -88.9809,Z 174,A -135.1031,B 7.8974,C 0.3238,E1 7.7867,E2 226.6488} C_DIS
LIN {X -95.5158,Y -92.0628,Z 174,A -133.2861,B 7.8972,C 0.3276,E1 7.7902,E2 224.8329} C_DIS
LIN {X -92.6434,Y -94.953,Z 174,A -131.5292,B 7.8971,C 0.331,E1 7.7936,E2 223.0769} C_DIS
LIN {X -90.1932,Y -97.2832,Z 174,A -129.9153,B 7.8971,C 0.3315,E1 7.797,E2 221.4446} C_DIS
LIN {X -86.7607,Y -100.3563,Z 174,A -128.0113,B 7.8969,C 0.3365,E1 7.8009,E2 219.5515} C_DIS
LIN {X -84.0505,Y -102.6366,Z 174,A -126.4945,B 7.8967,C 0.3393,E1 7.8042,E2 218.0367} C_DIS
LIN {X -80.973,Y -105.0821,Z 174,A -124.8664,B 7.8966,C 0.3433,E1 7.8078,E2 216.4174} C_DIS
LIN {X -78.8043,Y -106.7181,Z 174,A -123.6016,B 7.8966,C 0.3438,E1 7.8106,E2 215.1415} C_DIS
LIN {X -76.1456,Y -108.6312,Z 174,A -122.1971,B 7.8964,C 0.3462,E1 7.8138,E2 213.7385} C_DIS
LIN {X -73.4604,Y -110.4643,Z 174,A -120.7625,B 7.8964,C 0.3479,E1 7.8171,E2 212.3003} C_DIS
LIN {X -70.7313,Y -112.2312,Z 174,A -119.3264,B 7.8963,C 0.3494,E1 7.8205,E2 210.8604} C_DIS
LIN {X -67.9598,Y -113.9308,Z 174,A -117.9116,B 7.8963,C 0.3512,E1 7.8239,E2 209.4443} C_DIS
LIN {X -65.1478,Y -115.5618,Z 174,A -116.401,B 7.8963,C 0.3514,E1 7.8276,E2 207.9206} C_DIS
LIN {X -62.5273,Y -117.0008,Z 174,A -115.1687,B 7.8961,C 0.354,E1 7.8306,E2 206.6956} C_DIS
LIN {X -59.6424,Y -118.4963,Z 174,A -113.753,B 7.8961,C 0.3555,E1 7.8341,E2 205.2783} C_DIS
LIN {X -56.4572,Y -120.0477,Z 174,A -112.2307,B 7.8959,C 0.3574,E1 7.838,E2 203.757} C_DIS
LIN {X -53.7612,Y -121.2772,Z 174,A -110.9435,B 7.8959,C 0.3586,E1 7.8413,E2 202.4687} C_DIS
LIN {X -50.5014,Y -122.6715,Z 174,A -109.4021,B 7.8959,C 0.36,E1 7.8452,E2 200.926} C_DIS
LIN {X -47.7475,Y -123.7681,Z 174,A -108.0685,B 7.8959,C 0.3604,E1 7.8487,E2 199.5856} C_DIS
LIN {X -44.0063,Y -125.1481,Z 174,A -106.4737,B 7.8956,C 0.3639,E1 7.8529,E2 198.0063} C_DIS
LIN {X -40.9416,Y -126.184,Z 174,A -104.7881,B 7.8958,C 0.3604,E1 7.8574,E2 196.2848} C_DIS
LIN {X -36.9932,Y -127.3965,Z 174,A -103.1912,B 7.8956,C 0.3647,E1 7.8616,E2 194.7107} C_DIS
LIN {X -33.1959,Y -128.4393,Z 174,A -101.3199,B 7.8956,C 0.363,E1 7.8668,E2 192.8179} C_DIS
LIN {X -29.0627,Y -129.4368,Z 174,A -99.6436,B 7.8956,C 0.3666,E1 7.8713,E2 191.1609} C_DIS
LIN {X -25.5963,Y -130.1677,Z 174,A -98.147,B 7.8955,C 0.3678,E1 7.8753,E2 189.6681} C_DIS
LIN {X -22.682,Y -130.707,Z 174,A -96.7414,B 7.8955,C 0.3662,E1 7.8793,E2 188.2466} C_DIS
LIN {X -19.1807,Y -131.2654,Z 174,A -95.2785,B 7.8955,C 0.3679,E1 7.8833,E2 186.7916} C_DIS
LIN {X -15.9469,Y -131.6969,Z 174,A -93.8706,B 7.8955,C 0.3682,E1 7.8872,E2 185.3834} C_DIS
LIN {X -12.7159,Y -132.0479,Z 174,A -92.47,B 7.8955,C 0.3685,E1 7.8911,E2 183.9825} C_DIS
LIN {X -8.8907,Y -132.3626,Z 174,A -90.6238,B 7.8955,C 0.3655,E1 7.8963,E2 182.1124} C_DIS
LIN {X -4.8944,Y -132.5688,Z 174,A -89.0935,B 7.8955,C 0.3689,E1 7.9005,E2 180.6058} C_DIS
LIN {X -1.3346,Y -132.6535,Z 174,A -87.6251,B 7.8954,C 0.3699,E1 7.9046,E2 179.1454} C_DIS
LIN {X 0.9609,Y -132.6531,Z 174,A -86.8212,B 7.8952,C 0.373,E1 7.9068,E2 178.3641} C_DIS
Enddeposition()
LIN {X 0.9609,Y -132.6531,Z 174,A -86.8212,B 7.8952,C 0.373,E1 7.9068,E2 178.3641} C_DIS
Startdeposition()
$VEL.CP = VEL_PRINT
LIN {X 0.0558,Y -133.5678,Z 174,A -87.7354,B 7.8945,C 0.3866,E1 7.9038,E2 179.3772} C_DIS
LIN {X -4.127,Y -133.5028,Z 174,A -89.3141,B 7.8947,C 0.3831,E1 7.8995,E2 180.9299} C_DIS
LIN {X -7.9327,Y -133.3304,Z 174,A -91.0111,B 7.8947,C 0.3841,E1 7.8947,E2 182.6354} C_DIS
LIN {X -11.4605,Y -133.0735,Z 174,A -92.4222,B 7.8947,C 0.3821,E1 7.8908,E2 184.0341} C_DIS
LIN {X -14.4719,Y -132.7796,Z 174,A -93.8532,B 7.8947,C 0.3841,E1 7.8868,E2 185.4819} C_DIS
LIN {X -17.9965,Y -132.3494,Z 174,A -95.29,B 7.8947,C 0.3823,E1 7.8829,E2 186.9087} C_DIS
LIN {X -21.72,Y -131.7882,Z 174,A -97.0348,B 7.8947,C 0.3839,E1 7.878,E2 188.6699} C_DIS
LIN {X -26.0628,Y -130.9995,Z 174,A -98.9268,B 7.8947,C 0.3831,E1 7.8728,E2 190.5623} C_DIS
LIN {X -29.6875,Y -130.2246,Z 174,A -100.4364,B 7.8947,C 0.381,E1 7.8687,E2 192.0624} C_DIS
LIN {X -33.0839,Y -129.4036,Z 174,A -102.0118,B 7.8947,C 0.3814,E1 7.8644,E2 193.6476} C_DIS
LIN {X -39.0707,Y -127.7233,Z 174,A -105.0669,B 7.8945,C 0.3857,E1 7.8561,E2 196.7508} C_DIS
LIN {X -43.0335,Y -126.4454,Z 174,A -106.383,B 7.895,C 0.3768,E1 7.8528,E2 198.0096} C_DIS
LIN {X -47.6056,Y -124.7961,Z 174,A -108.497,B 7.895,C 0.3754,E1 7.8472,E2 200.1275} C_DIS
LIN {X -50.8977,Y -123.489,Z 174,A -109.966,B 7.8951,C 0.3732,E1 7.8434,E2 201.5904} C_DIS
LIN {X -54.7241,Y -121.8402,Z 174,A -111.8812,B 7.8951,C 0.3732,E1 7.8385,E2 203.5215} C_DIS
LIN {X -58.1369,Y -120.2506,Z 174,A -113.464,B 7.8952,C 0.371,E1 7.8345,E2 205.1005} C_DIS
LIN {X -60.8545,Y -118.8971,Z 174,A -114.8287,B 7.8952,C 0.3704,E1 7.8311,E2 206.4727} C_DIS
LIN {X -64.7621,Y -116.8166,Z 174,A -116.7806,B 7.8953,C 0.3688,E1 7.8263,E2 208.4311} C_DIS
LIN {X -68.2872,Y -114.7917,Z 174,A -118.5456,B 7.8954,C 0.3667,E1 7.822,E2 210.1987} C_DIS
LIN {X -71.6844,Y -112.7021,Z 174,A -120.3232,B 7.8954,C 0.3653,E1 7.8178,E2 211.9844} C_DIS
LIN {X -75.0516,Y -110.4878,Z 174,A -121.9133,B 7.8957,C 0.3606,E1 7.8141,E2 213.5573} C_DIS
LIN {X -79.1515,Y -107.5885,Z 174,A -124.213,B 7.8957,C 0.3593,E1 7.8089,E2 215.8746} C_DIS
LIN {X -82.3497,Y -105.1609,Z 174,A -126.0377,B 7.8958,C 0.358,E1 7.8048,E2 217.7115} C_DIS
LIN {X -85.7403,Y -102.4152,Z 174,A -127.8328,B 7.896,C 0.3536,E1 7.801,E2 219.4969} C_DIS
LIN {X -89.14,Y -99.4702,Z 174,A -129.9385,B 7.896,C 0.3526,E1 7.7965,E2 221.6236} C_DIS
LIN {X -91.9754,Y -96.8554,Z 174,A -131.501,B 7.8963,C 0.3481,E1 7.7934,E2 223.1744} C_DIS
LIN {X -94.5423,Y -94.3509,Z 174,A -133.0178,B 7.8964,C 0.3448,E1 7.7904,E2 224.6882} C_DIS
LIN {X -98.0184,Y -90.7348,Z 174,A -135.1201,B 7.8966,C 0.3398,E1 7.7863,E2 226.7838} C_DIS
LIN {X -100.7277,Y -87.7165,Z 174,A -136.9364,B 7.8967,C 0.3372,E1 7.783,E2 228.6088} C_DIS
LIN {X -103.552,Y -84.3639,Z 174,A -138.942,B 7.8968,C 0.335,E1 7.7794,E2 230.6289} C_DIS
LIN {X -106.3889,Y -80.7576,Z 174,A -140.8892,B 7.897,C 0.3303,E1 7.776,E2 232.5727} C_DIS
LIN {X -108.8118,Y -77.4618,Z 174,A -142.629,B 7.8972,C 0.3261,E1 7.7732,E2 234.3099} C_DIS
LIN {X -111.2318,Y -73.9446,Z 174,A -144.5038,B 7.8973,C 0.3224,E1 7.7703,E2 236.1892} C_DIS
LIN {X -113.6489,Y -70.1736,Z 174,A -146.5001,B 7.8975,C 0.3189,E1 7.7673,E2 238.1936} C_DIS
LIN {X -117.4393,Y -63.6271,Z 174,A -149.8143,B 7.8978,C 0.3119,E1 7.7627,E2 241.5145} C_DIS
LIN {X -119.2085,Y -60.2428,Z 174,A -151.4303,B 7.8979,C 0.3074,E1 7.7606,E2 243.1268} C_DIS
LIN {X -121.5392,Y -55.3938,Z 174,A -153.7118,B 7.8982,C 0.3011,E1 7.7579,E2 245.4038} C_DIS
LIN {X -123.213,Y -51.5586,Z 174,A -155.5353,B 7.8983,C 0.2968,E1 7.7559,E2 247.2296} C_DIS
LIN {X -124.575,Y -48.1752,Z 174,A -157.1117,B 7.8985,C 0.2928,E1 7.7543,E2 248.8064} C_DIS
LIN {X -125.9934,Y -44.3374,Z 174,A -158.7911,B 7.8987,C 0.2871,E1 7.7527,E2 250.4755} C_DIS
LIN {X -126.8617,Y -41.7858,Z 174,A -160.0621,B 7.8987,C 0.2855,E1 7.7516,E2 251.7595} C_DIS
LIN {X -128.2276,Y -37.3829,Z 174,A -162.339,B 7.8988,C 0.2842,E1 7.7497,E2 254.071} C_DIS
LIN {X -130.1659,Y -29.9445,Z 174,A -165.354,B 7.8993,C 0.2712,E1 7.7477,E2 257.0497} C_DIS
LIN {X -131.3164,Y -24.4184,Z 174,A -167.8419,B 7.8995,C 0.2653,E1 7.7463,E2 259.5439} C_DIS
LIN {X -131.781,Y -21.7628,Z 174,A -169.0242,B 7.8995,C 0.2624,E1 7.7457,E2 260.7283} C_DIS
LIN {X -132.2578,Y -18.6482,Z 174,A -170.4655,B 7.8996,C 0.2597,E1 7.7451,E2 262.1793} C_DIS
LIN {X -132.7794,Y -14.4738,Z 174,A -172.3062,B 7.8998,C 0.2551,E1 7.7445,E2 264.0228} C_DIS
LIN {X -133.0881,Y -11.287,Z 174,A -173.7482,B 7.8998,C 0.252,E1 7.7442,E2 265.4719} C_DIS
LIN {X -133.3663,Y -7.3254,Z 174,A -175.5475,B 7.9,C 0.2484,E1 7.7439,E2 267.2812} C_DIS
LIN {X -133.5239,Y -3.3705,Z 174,A -177.2851,B 7.9001,C 0.2441,E1 7.7437,E2 269.0221} C_DIS
LIN {X -133.5654,Y 0.6823,Z 174,A -179.0204,B 7.9003,C 0.239,E1 7.7437,E2 270.7555} C_DIS
LIN {X -133.4754,Y 4.9242,Z 174,A 179.1562,B 7.9004,C 0.2338,E1 7.7438,E2 272.5778} C_DIS
LIN {X -133.2904,Y 8.5831,Z 174,A 177.6869,B 7.9006,C 0.2279,E1 7.7441,E2 274.0334} C_DIS
LIN {X -133.0641,Y 11.5715,Z 174,A 176.2322,B 7.9006,C 0.2265,E1 7.7444,E2 275.5072} C_DIS
LIN {X -132.635,Y 15.7413,Z 174,A 174.5212,B 7.9008,C 0.2201,E1 7.7449,E2 277.206} C_DIS
LIN {X -132.2213,Y 18.9035,Z 174,A 173.0346,B 7.9009,C 0.2178,E1 7.7455,E2 278.7055} C_DIS
LIN {X -131.5396,Y 23.1791,Z 174,A 171.1346,B 7.901,C 0.2131,E1 7.7464,E2 280.6089} C_DIS
LIN {X -130.8584,Y 26.7559,Z 174,A 169.5836,B 7.9012,C 0.2085,E1 7.7472,E2 282.1571} C_DIS
LIN {X -129.9561,Y 30.845,Z 174,A 167.7236,B 7.9012,C 0.2043,E1 7.7484,E2 284.023} C_DIS
LIN {X -129.0389,Y 34.4781,Z 174,A 166.0637,B 7.9014,C 0.2005,E1 7.7495,E2 285.6875} C_DIS
LIN {X -128.0988,Y 37.8226,Z 174,A 164.5796,B 7.9014,C 0.1962,E1 7.7507,E2 287.1695} C_DIS
LIN {X -126.9861,Y 41.4118,Z 174,A 162.9832,B 7.9016,C 0.1916,E1 7.752,E2 288.7626} C_DIS
LIN {X -125.3815,Y 46.0414,Z 174,A 160.6415,B 7.9016,C 0.1891,E1 7.7542,E2 291.1307} C_DIS
LIN {X -124.174,Y 49.2053,Z 174,A 159.3743,B 7.9018,C 0.1827,E1 7.7555,E2 292.3745} C_DIS
LIN {X -123.1477,Y 51.7149,Z 174,A 158.1707,B 7.9018,C 0.1801,E1 7.7568,E2 293.5817} C_DIS
LIN {X -121.8784,Y 54.6387,Z 174,A 156.7569,B 7.9019,C 0.1771,E1 7.7584,E2 294.9996} C_DIS
LIN {X -120.383,Y 57.8598,Z 174,A 155.2912,B 7.902,C 0.1723,E1 7.7601,E2 296.457} C_DIS
LIN {X -119.0357,Y 60.5823,Z 174,A 153.8693,B 7.902,C 0.1705,E1 7.7619,E2 297.8918} C_DIS
LIN {X -116.9934,Y 64.4422,Z 174,A 151.6072,B 7.902,C 0.171,E1 7.765,E2 300.198} C_DIS
LIN {X -115.1713,Y 67.6449,Z 174,A 149.8104,B 7.902,C 0.17,E1 7.7676,E2 302.0186} C_DIS
LIN {X -112.7247,Y 71.649,Z 174,A 148.3654,B 7.9023,C 0.1573,E1 7.7696,E2 303.3948} C_DIS
LIN {X -109.0377,Y 77.1431,Z 174,A 145.4672,B 7.9024,C 0.1513,E1 7.7742,E2 306.2973} C_DIS
LIN {X -106.8317,Y 80.1709,Z 174,A 143.8238,B 7.9025,C 0.1481,E1 7.7769,E2 307.9435} C_DIS
LIN {X -104.3595,Y 83.363,Z 174,A 141.977,B 7.9025,C 0.1457,E1 7.7801,E2 309.8022} C_DIS
LIN {X -101.4879,Y 86.8367,Z 174,A 139.9938,B 7.9026,C 0.1421,E1 7.7837,E2 311.7895} C_DIS
LIN {X -98.5707,Y 90.1343,Z 174,A 138.0578,B 7.9026,C 0.1387,E1 7.7873,E2 313.7293} C_DIS
LIN {X -95.406,Y 93.477,Z 174,A 136.0489,B 7.9027,C 0.135,E1 7.7912,E2 315.7404} C_DIS
LIN {X -92.0474,Y 96.7865,Z 174,A 134.0472,B 7.9028,C 0.1307,E1 7.7952,E2 317.7377} C_DIS
LIN {X -88.9259,Y 99.6619,Z 174,A 132.1862,B 7.9028,C 0.1277,E1 7.7991,E2 319.6018} C_DIS
LIN {X -85.5243,Y 102.5964,Z 174,A 130.2423,B 7.9029,C 0.1243,E1 7.8032,E2 321.5459} C_DIS
LIN {X -82.3293,Y 105.1769,Z 174,A 128.4844,B 7.9029,C 0.1211,E1 7.807,E2 323.3018} C_DIS
LIN {X -78.8335,Y 107.8222,Z 174,A 126.3884,B 7.9029,C 0.1209,E1 7.8118,E2 325.4214} C_DIS
LIN {X -75.148,Y 110.4226,Z 174,A 124.7348,B 7.9031,C 0.1136,E1 7.8155,E2 327.0403} C_DIS
LIN {X -71.514,Y 112.8099,Z 174,A 123.0457,B 7.9031,C 0.1081,E1 7.8194,E2 328.7071} C_DIS
LIN {X -69.1356,Y 114.2826,Z 174,A 121.5303,B 7.9031,C 0.1109,E1 7.8231,E2 330.2587} C_DIS
LIN {X -65.3129,Y 116.5097,Z 174,A 119.6212,B 7.9031,C 0.1083,E1 7.8277,E2 332.1675} C_DIS
LIN {X -61.4741,Y 118.5797,Z 174,A 117.8334,B 7.9031,C 0.1046,E1 7.8321,E2 333.9441} C_DIS
LIN {X -58.1078,Y 120.2645,Z 174,A 116.275,B 7.9032,C 0.1016,E1 7.836,E2 335.4944} C_DIS
LIN {X -55.3002,Y 121.5825,Z 174,A 114.8385,B 7.9032,C 0.1016,E1 7.8397,E2 336.9425} C_DIS
LIN {X -52.2804,Y 122.911,Z 174,A 112.7804,B 7.9032,C 0.1096,E1 7.8451,E2 339.0748} C_DIS
LIN {X -47.7187,Y 124.7525,Z 174,A 111.3178,B 7.9032,C 0.0976,E1 7.8487,E2 340.46} C_DIS
LIN {X -43.6304,Y 126.2385,Z 174,A 109.4041,B 7.9032,C 0.0965,E1 7.8538,E2 342.378} C_DIS
LIN {X -40.5323,Y 127.2671,Z 174,A 108.0258,B 7.9033,C 0.0949,E1 7.8574,E2 343.7527} C_DIS
LIN {X -35.4334,Y 128.7811,Z 174,A 105.7511,B 7.9033,C 0.093,E1 7.8635,E2 346.0251} C_DIS
Enddeposition()
END
